gfCNCPoint5[9670] = {X 422.3701, Y 16.1525, Z -7.1667, A 0.000, B 0.000, C 0.000 }
gfCNCPoint5[9671] = {X 421.6779, Y 16.7020, Z -7.1667, A 0.000, B 0.000, C 0.000 }
gfCNCPoint5[9672] = {X 420.8909, Y 17.1044, Z -7.1667, A 0.000, B 0.000, C 0.000 }
gfCNCPoint5[9673] = {X 420.1838, Y 18.0570, Z -7.1667, A 0.000, B 0.000, C 0.000 }
gfCNCPoint5[9674] = {X 419.5438, Y 19.0559, Z -7.1667, A 0.000, B 0.000, C 0.000 }
gfCNCPoint5[9675] = {X 418.0618, Y 21.4548, Z -7.1667, A 0.000, B 0.000, C 0.000 }
gfCNCPoint5[9676] = {X 411.6279, Y 31.7882, Z -7.1667, A 0.000, B 0.000, C 0.000 }
gfCNCPoint5[9677] = {X 411.6285, Y 40.8613, Z -7.1667, A 0.000, B 0.000, C 0.000 }
gfCNCPoint5[9678] = {X 412.2676, Y 41.5581, Z -7.1667, A 0.000, B 0.000, C 0.000 }
gfCNCPoint5[9679] = {X 412.7477, Y 42.3727, Z -7.1667, A 0.000, B 0.000, C 0.000 }
gfCNCPoint5[9680] = {X 413.0478, Y 43.2694, Z -7.1667, A 0.000, B 0.000, C 0.000 }
gfCNCPoint5[9681] = {X 413.1547, Y 44.2088, Z -7.1667, A 0.000, B 0.000, C 0.000 }
gfCNCPoint5[9682] = {X 413.1545, Y 45.0423, Z -7.1667, A 0.000, B 0.000, C 0.000 }
gfCNCPoint5[9683] = {X 413.0719, Y 45.8494, Z -7.1667, A 0.000, B 0.000, C 0.000 }
gfCNCPoint5[9684] = {X 412.8426, Y 46.6276, Z -7.1667, A 0.000, B 0.000, C 0.000 }
gfCNCPoint5[9685] = {X 412.4743, Y 47.3505, Z -7.1667, A 0.000, B 0.000, C 0.000 }
gfCNCPoint5[9686] = {X 411.9795, Y 47.9934, Z -7.1667, A 0.000, B 0.000, C 0.000 }
gfCNCPoint5[9687] = {X 412.3313, Y 48.3200, Z -7.1667, A 0.000, B 0.000, C 0.000 }
gfCNCPoint5[9688] = {X 419.4886, Y 48.3200, Z -7.1667, A 0.000, B 0.000, C 0.000 }
gfCNCPoint5[9689] = {X 420.8006, Y 48.4093, Z -7.1667, A 0.000, B 0.000, C 0.000 }
gfCNCPoint5[9690] = {X 422.0883, Y 48.6756, Z -7.1667, A 0.000, B 0.000, C 0.000 }
gfCNCPoint5[9691] = {X 423.3281, Y 49.1140, Z -7.1667, A 0.000, B 0.000, C 0.000 }
gfCNCPoint5[9692] = {X 424.4970, Y 49.7164, Z -7.1667, A 0.000, B 0.000, C 0.000 }
gfCNCPoint5[9693] = {X 425.4625, Y 50.3832, Z -7.1667, A 0.000, B 0.000, C 0.000 }
gfCNCPoint5[9694] = {X 426.3402, Y 51.1620, Z -7.1667, A 0.000, B 0.000, C 0.000 }
gfCNCPoint5[9695] = {X 427.1172, Y 52.0412, Z -7.1667, A 0.000, B 0.000, C 0.000 }
gfCNCPoint5[9696] = {X 427.7821, Y 53.0080, Z -7.1667, A 0.000, B 0.000, C 0.000 }
gfCNCPoint5[9697] = {X 428.1265, Y 53.6309, Z -7.1667, A 0.000, B 0.000, C 0.000 }
gfCNCPoint5[9698] = {X 428.4242, Y 54.2773, Z -7.1667, A 0.000, B 0.000, C 0.000 }
gfCNCPoint5[9699] = {X 431.5822, Y 55.5078, Z -7.1667, A 0.000, B 0.000, C 0.000 }
gfCNCPoint5[9700] = {X 439.8795, Y 58.7999, Z -7.1667, A 0.000, B 0.000, C 0.000 }
gfCNCPoint5[9701] = {X 441.6498, Y 54.3383, Z -7.1667, A 0.000, B 0.000, C 0.000 }
gfCNCPoint5[9702] = {X 444.2225, Y 55.3591, Z -7.1667, A 0.000, B 0.000, C 0.000 }
gfCNCPoint5[9703] = {X 444.5427, Y 54.0013, Z -7.1667, A 0.000, B 0.000, C 0.000 }
gfCNCPoint5[9704] = {X 444.9921, Y 52.6806, Z -7.1667, A 0.000, B 0.000, C 0.000 }
gfCNCPoint5[9705] = {X 443.9527, Y 53.3760, Z -7.1667, A 0.000, B 0.000, C 0.000 }
gfCNCPoint5[9706] = {X 442.8324, Y 53.9317, Z -7.1667, A 0.000, B 0.000, C 0.000 }
gfCNCPoint5[9707] = {X 441.6498, Y 54.3383, Z -7.1667, A 0.000, B 0.000, C 0.000 }
gfCNCPoint5[9708] = {X 440.7647, Y 56.5691, Z -7.1667, A 0.000, B 0.000, C 0.000 }
gfCNCPoint5[9709] = {X 446.3797, Y 58.7970, Z -7.1667, A 0.000, B 0.000, C 0.000 }
gfCNCPoint5[9710] = {X 446.3796, Y 58.0000, Z -7.1667, A 0.000, B 0.000, C 0.000 }
gfCNCPoint5[9711] = {X 446.4304, Y 56.8937, Z -7.1667, A 0.000, B 0.000, C 0.000 }
gfCNCPoint5[9712] = {X 446.5822, Y 55.7968, Z -7.1667, A 0.000, B 0.000, C 0.000 }
gfCNCPoint5[9713] = {X 446.8494, Y 54.6640, Z -7.1667, A 0.000, B 0.000, C 0.000 }
gfCNCPoint5[9714] = {X 447.2243, Y 53.5622, Z -7.1667, A 0.000, B 0.000, C 0.000 }
gfCNCPoint5[9715] = {X 447.8767, Y 52.1752, Z -7.1667, A 0.000, B 0.000, C 0.000 }
gfCNCPoint5[9716] = {X 448.6995, Y 50.8820, Z -7.1667, A 0.000, B 0.000, C 0.000 }
gfCNCPoint5[9717] = {X 447.8224, Y 50.1272, Z -7.1667, A 0.000, B 0.000, C 0.000 }
gfCNCPoint5[9718] = {X 447.0760, Y 49.2431, Z -7.1667, A 0.000, B 0.000, C 0.000 }
gfCNCPoint5[9719] = {X 446.4792, Y 48.2518, Z -7.1667, A 0.000, B 0.000, C 0.000 }
gfCNCPoint5[9720] = {X 446.0469, Y 47.1785, Z -7.1667, A 0.000, B 0.000, C 0.000 }
gfCNCPoint5[9721] = {X 445.6333, Y 48.2126, Z -7.1667, A 0.000, B 0.000, C 0.000 }
gfCNCPoint5[9722] = {X 445.0668, Y 49.1715, Z -7.1667, A 0.000, B 0.000, C 0.000 }
gfCNCPoint5[9723] = {X 444.3606, Y 50.0328, Z -7.1667, A 0.000, B 0.000, C 0.000 }
gfCNCPoint5[9724] = {X 443.5314, Y 50.7763, Z -7.1667, A 0.000, B 0.000, C 0.000 }
gfCNCPoint5[9725] = {X 442.7497, Y 51.2993, Z -7.1667, A 0.000, B 0.000, C 0.000 }
gfCNCPoint5[9726] = {X 441.9071, Y 51.7172, Z -7.1667, A 0.000, B 0.000, C 0.000 }
gfCNCPoint5[9727] = {X 441.0177, Y 52.0230, Z -7.1667, A 0.000, B 0.000, C 0.000 }
gfCNCPoint5[9728] = {X 440.0677, Y 52.2155, Z -7.1667, A 0.000, B 0.000, C 0.000 }
gfCNCPoint5[9729] = {X 439.1005, Y 52.2800, Z -7.1667, A 0.000, B 0.000, C 0.000 }
gfCNCPoint5[9730] = {X 432.5144, Y 52.2800, Z -7.1667, A 0.000, B 0.000, C 0.000 }
gfCNCPoint5[9731] = {X 431.6034, Y 52.2228, Z -7.1667, A 0.000, B 0.000, C 0.000 }
gfCNCPoint5[9732] = {X 430.7066, Y 52.0520, Z -7.1667, A 0.000, B 0.000, C 0.000 }
gfCNCPoint5[9733] = {X 429.8384, Y 51.7703, Z -7.1667, A 0.000, B 0.000, C 0.000 }
gfCNCPoint5[9734] = {X 430.0166, Y 52.0766, Z -7.1667, A 0.000, B 0.000, C 0.000 }
gfCNCPoint5[9735] = {X 430.1859, Y 52.3880, Z -7.1667, A 0.000, B 0.000, C 0.000 }
gfCNCPoint5[9736] = {X 432.4639, Y 53.2756, Z -7.1667, A 0.000, B 0.000, C 0.000 }
gfCNCPoint5[9737] = {X 440.7647, Y 56.5691, Z -7.1667, A 0.000, B 0.000, C 0.000 }
gfCNCPoint5[9738] = {X 439.8795, Y 58.7999, Z -7.1667, A 0.000, B 0.000, C 0.000 }
gfCNCPoint5[9739] = {X 449.5091, Y 62.6207, Z -7.1667, A 0.000, B 0.000, C 0.000 }
gfCNCPoint5[9740] = {X 449.1112, Y 61.4460, Z -7.1667, A 0.000, B 0.000, C 0.000 }
gfCNCPoint5[9741] = {X 448.8668, Y 60.2301, Z -7.1667, A 0.000, B 0.000, C 0.000 }
gfCNCPoint5[9742] = {X 448.7798, Y 58.9930, Z -7.1667, A 0.000, B 0.000, C 0.000 }
gfCNCPoint5[9743] = {X 448.7796, Y 58.0000, Z -7.1667, A 0.000, B 0.000, C 0.000 }
gfCNCPoint5[9744] = {X 448.8564, Y 56.7833, Z -7.1667, A 0.000, B 0.000, C 0.000 }
gfCNCPoint5[9745] = {X 449.0855, Y 55.5859, Z -7.1667, A 0.000, B 0.000, C 0.000 }
gfCNCPoint5[9746] = {X 449.4632, Y 54.4268, Z -7.1667, A 0.000, B 0.000, C 0.000 }
gfCNCPoint5[9747] = {X 449.9837, Y 53.3244, Z -7.1667, A 0.000, B 0.000, C 0.000 }
gfCNCPoint5[9748] = {X 450.6386, Y 52.2961, Z -7.1667, A 0.000, B 0.000, C 0.000 }
gfCNCPoint5[9749] = {X 451.3887, Y 51.3890, Z -7.1667, A 0.000, B 0.000, C 0.000 }
gfCNCPoint5[9750] = {X 452.2434, Y 50.5796, Z -7.1667, A 0.000, B 0.000, C 0.000 }
gfCNCPoint5[9751] = {X 453.1901, Y 49.8800, Z -7.1667, A 0.000, B 0.000, C 0.000 }
gfCNCPoint5[9752] = {X 452.3731, Y 49.8442, Z -7.1667, A 0.000, B 0.000, C 0.000 }
gfCNCPoint5[9753] = {X 451.5735, Y 49.6724, Z -7.1667, A 0.000, B 0.000, C 0.000 }
gfCNCPoint5[9754] = {X 450.8138, Y 49.3696, Z -7.1667, A 0.000, B 0.000, C 0.000 }
gfCNCPoint5[9755] = {X 450.1154, Y 48.9441, Z -7.1667, A 0.000, B 0.000, C 0.000 }
gfCNCPoint5[9756] = {X 449.3503, Y 48.2496, Z -7.1667, A 0.000, B 0.000, C 0.000 }
gfCNCPoint5[9757] = {X 448.7486, Y 47.4095, Z -7.1667, A 0.000, B 0.000, C 0.000 }
gfCNCPoint5[9758] = {X 448.3373, Y 46.4616, Z -7.1667, A 0.000, B 0.000, C 0.000 }
gfCNCPoint5[9759] = {X 448.1732, Y 45.7588, Z -7.1667, A 0.000, B 0.000, C 0.000 }
gfCNCPoint5[9760] = {X 448.1146, Y 45.0395, Z -7.1667, A 0.000, B 0.000, C 0.000 }
gfCNCPoint5[9761] = {X 448.1149, Y 44.1417, Z -7.1667, A 0.000, B 0.000, C 0.000 }
gfCNCPoint5[9762] = {X 448.2252, Y 43.1751, Z -7.1667, A 0.000, B 0.000, C 0.000 }
gfCNCPoint5[9763] = {X 448.5250, Y 42.2497, Z -7.1667, A 0.000, B 0.000, C 0.000 }
gfCNCPoint5[9764] = {X 449.0024, Y 41.4021, Z -7.1667, A 0.000, B 0.000, C 0.000 }
gfCNCPoint5[9765] = {X 449.6384, Y 40.6660, Z -7.1667, A 0.000, B 0.000, C 0.000 }
gfCNCPoint5[9766] = {X 449.6384, Y 35.0338, Z -7.1667, A 0.000, B 0.000, C 0.000 }
gfCNCPoint5[9767] = {X 447.8174, Y 35.0338, Z -7.1667, A 0.000, B 0.000, C 0.000 }
gfCNCPoint5[9768] = {X 443.7931, Y 42.8695, Z -7.1667, A 0.000, B 0.000, C 0.000 }
gfCNCPoint5[9769] = {X 443.9303, Y 43.5111, Z -7.1667, A 0.000, B 0.000, C 0.000 }
gfCNCPoint5[9770] = {X 443.9803, Y 44.1653, Z -7.1667, A 0.000, B 0.000, C 0.000 }
gfCNCPoint5[9771] = {X 443.9805, Y 45.0000, Z -7.1667, A 0.000, B 0.000, C 0.000 }
gfCNCPoint5[9772] = {X 443.9242, Y 45.7387, Z -7.1667, A 0.000, B 0.000, C 0.000 }
gfCNCPoint5[9773] = {X 443.7568, Y 46.4603, Z -7.1667, A 0.000, B 0.000, C 0.000 }
gfCNCPoint5[9774] = {X 443.3474, Y 47.4038, Z -7.1667, A 0.000, B 0.000, C 0.000 }
gfCNCPoint5[9775] = {X 442.7493, Y 48.2405, Z -7.1667, A 0.000, B 0.000, C 0.000 }
gfCNCPoint5[9776] = {X 441.9891, Y 48.9332, Z -7.1667, A 0.000, B 0.000, C 0.000 }
gfCNCPoint5[9777] = {X 441.1006, Y 49.4513, Z -7.1667, A 0.000, B 0.000, C 0.000 }
gfCNCPoint5[9778] = {X 440.1232, Y 49.7716, Z -7.1667, A 0.000, B 0.000, C 0.000 }
gfCNCPoint5[9779] = {X 439.1005, Y 49.8800, Z -7.1667, A 0.000, B 0.000, C 0.000 }
gfCNCPoint5[9780] = {X 432.5144, Y 49.8800, Z -7.1667, A 0.000, B 0.000, C 0.000 }
gfCNCPoint5[9781] = {X 431.6014, Y 49.7938, Z -7.1667, A 0.000, B 0.000, C 0.000 }
gfCNCPoint5[9782] = {X 430.7206, Y 49.5383, Z -7.1667, A 0.000, B 0.000, C 0.000 }
gfCNCPoint5[9783] = {X 429.8343, Y 49.0782, Z -7.1667, A 0.000, B 0.000, C 0.000 }
gfCNCPoint5[9784] = {X 429.0603, Y 48.4473, Z -7.1667, A 0.000, B 0.000, C 0.000 }
gfCNCPoint5[9785] = {X 428.4309, Y 47.6720, Z -7.1667, A 0.000, B 0.000, C 0.000 }
gfCNCPoint5[9786] = {X 427.9725, Y 46.7848, Z -7.1667, A 0.000, B 0.000, C 0.000 }
gfCNCPoint5[9787] = {X 427.7197, Y 45.9083, Z -7.1667, A 0.000, B 0.000, C 0.000 }
gfCNCPoint5[9788] = {X 427.6344, Y 45.0000, Z -7.1667, A 0.000, B 0.000, C 0.000 }
gfCNCPoint5[9789] = {X 427.6344, Y 44.2089, Z -7.1667, A 0.000, B 0.000, C 0.000 }
gfCNCPoint5[9790] = {X 427.7263, Y 43.2661, Z -7.1667, A 0.000, B 0.000, C 0.000 }
gfCNCPoint5[9791] = {X 427.9987, Y 42.3588, Z -7.1667, A 0.000, B 0.000, C 0.000 }
gfCNCPoint5[9792] = {X 428.4412, Y 41.5212, Z -7.1667, A 0.000, B 0.000, C 0.000 }
gfCNCPoint5[9793] = {X 429.0371, Y 40.7849, Z -7.1667, A 0.000, B 0.000, C 0.000 }
gfCNCPoint5[9794] = {X 429.7641, Y 40.1776, Z -7.1667, A 0.000, B 0.000, C 0.000 }
gfCNCPoint5[9795] = {X 430.5947, Y 39.7222, Z -7.1667, A 0.000, B 0.000, C 0.000 }
gfCNCPoint5[9796] = {X 434.2527, Y 32.5621, Z -7.1667, A 0.000, B 0.000, C 0.000 }
gfCNCPoint5[9797] = {X 432.9253, Y 31.5659, Z -7.1667, A 0.000, B 0.000, C 0.000 }
gfCNCPoint5[9798] = {X 431.7497, Y 30.3944, Z -7.1667, A 0.000, B 0.000, C 0.000 }
gfCNCPoint5[9799] = {X 430.7488, Y 29.0705, Z -7.1667, A 0.000, B 0.000, C 0.000 }
gfCNCPoint5[9800] = {X 429.9422, Y 27.6200, Z -7.1667, A 0.000, B 0.000, C 0.000 }
gfCNCPoint5[9801] = {X 429.3457, Y 26.0712, Z -7.1667, A 0.000, B 0.000, C 0.000 }
gfCNCPoint5[9802] = {X 428.8989, Y 24.1613, Z -7.1667, A 0.000, B 0.000, C 0.000 }
gfCNCPoint5[9803] = {X 428.6737, Y 22.2128, Z -7.1667, A 0.000, B 0.000, C 0.000 }
gfCNCPoint5[9804] = {X 428.6731, Y 20.2514, Z -7.1667, A 0.000, B 0.000, C 0.000 }
gfCNCPoint5[9805] = {X 428.8972, Y 18.3027, Z -7.1667, A 0.000, B 0.000, C 0.000 }
gfCNCPoint5[9806] = {X 429.3429, Y 16.3926, Z -7.1667, A 0.000, B 0.000, C 0.000 }
gfCNCPoint5[9807] = {X 429.8636, Y 14.9601, Z -7.1667, A 0.000, B 0.000, C 0.000 }
gfCNCPoint5[9808] = {X 430.5563, Y 13.6023, Z -7.1667, A 0.000, B 0.000, C 0.000 }
gfCNCPoint5[9809] = {X 431.4105, Y 12.3399, Z -7.1667, A 0.000, B 0.000, C 0.000 }
gfCNCPoint5[9810] = {X 432.4132, Y 11.1919, Z -7.1667, A 0.000, B 0.000, C 0.000 }
gfCNCPoint5[9811] = {X 433.5448, Y 10.1793, Z -7.1667, A 0.000, B 0.000, C 0.000 }
gfCNCPoint5[9812] = {X 434.7918, Y 9.3127, Z -7.1667, A 0.000, B 0.000, C 0.000 }
gfCNCPoint5[9813] = {X 436.1354, Y 8.6052, Z -7.1667, A 0.000, B 0.000, C 0.000 }
gfCNCPoint5[9814] = {X 437.5555, Y 8.0674, Z -7.1667, A 0.000, B 0.000, C 0.000 }
gfCNCPoint5[9815] = {X 439.0308, Y 7.7073, Z -7.1667, A 0.000, B 0.000, C 0.000 }
gfCNCPoint5[9816] = {X 441.1775, Y 7.4101, Z -7.1667, A 0.000, B 0.000, C 0.000 }
gfCNCPoint5[9817] = {X 443.3425, Y 7.3136, Z -7.1667, A 0.000, B 0.000, C 0.000 }
gfCNCPoint5[9818] = {X 459.4469, Y 7.3096, Z -7.1667, A 0.000, B 0.000, C 0.000 }
gfCNCPoint5[9819] = {X 460.4098, Y 7.4057, Z -7.1667, A 0.000, B 0.000, C 0.000 }
gfCNCPoint5[9820] = {X 461.3347, Y 7.6903, Z -7.1667, A 0.000, B 0.000, C 0.000 }
gfCNCPoint5[9821] = {X 462.1851, Y 8.1521, Z -7.1667, A 0.000, B 0.000, C 0.000 }
gfCNCPoint5[9822] = {X 462.9274, Y 8.7728, Z -7.1667, A 0.000, B 0.000, C 0.000 }
gfCNCPoint5[9823] = {X 463.5324, Y 9.5281, Z -7.1667, A 0.000, B 0.000, C 0.000 }
gfCNCPoint5[9824] = {X 463.9761, Y 10.3881, Z -7.1667, A 0.000, B 0.000, C 0.000 }
gfCNCPoint5[9825] = {X 464.2317, Y 11.2682, Z -7.1667, A 0.000, B 0.000, C 0.000 }
gfCNCPoint5[9826] = {X 464.3179, Y 12.1806, Z -7.1667, A 0.000, B 0.000, C 0.000 }
gfCNCPoint5[9827] = {X 464.3179, Y 12.9780, Z -7.1667, A 0.000, B 0.000, C 0.000 }
gfCNCPoint5[9828] = {X 464.2174, Y 13.9633, Z -7.1667, A 0.000, B 0.000, C 0.000 }
gfCNCPoint5[9829] = {X 463.9200, Y 14.9081, Z -7.1667, A 0.000, B 0.000, C 0.000 }
gfCNCPoint5[9830] = {X 463.4380, Y 15.7733, Z -7.1667, A 0.000, B 0.000, C 0.000 }
gfCNCPoint5[9831] = {X 462.7912, Y 16.5234, Z -7.1667, A 0.000, B 0.000, C 0.000 }
gfCNCPoint5[9832] = {X 462.7910, Y 16.7696, Z -7.1667, A 0.000, B 0.000, C 0.000 }
gfCNCPoint5[9833] = {X 462.7919, Y 40.6641, Z -7.1667, A 0.000, B 0.000, C 0.000 }
gfCNCPoint5[9834] = {X 463.4324, Y 41.4055, Z -7.1667, A 0.000, B 0.000, C 0.000 }
gfCNCPoint5[9835] = {X 463.9119, Y 42.2600, Z -7.1667, A 0.000, B 0.000, C 0.000 }
gfCNCPoint5[9836] = {X 464.2110, Y 43.1930, Z -7.1667, A 0.000, B 0.000, C 0.000 }
gfCNCPoint5[9837] = {X 464.3178, Y 44.1670, Z -7.1667, A 0.000, B 0.000, C 0.000 }
gfCNCPoint5[9838] = {X 464.3179, Y 45.0000, Z -7.1667, A 0.000, B 0.000, C 0.000 }
gfCNCPoint5[9839] = {X 464.3082, Y 45.3090, Z -7.1667, A 0.000, B 0.000, C 0.000 }
gfCNCPoint5[9840] = {X 464.2788, Y 45.6167, Z -7.1667, A 0.000, B 0.000, C 0.000 }
gfCNCPoint5[9841] = {X 464.0485, Y 46.5992, Z -7.1667, A 0.000, B 0.000, C 0.000 }
gfCNCPoint5[9842] = {X 463.6209, Y 47.5134, Z -7.1667, A 0.000, B 0.000, C 0.000 }
gfCNCPoint5[9843] = {X 463.0145, Y 48.3200, Z -7.1667, A 0.000, B 0.000, C 0.000 }
gfCNCPoint5[9844] = {X 462.6627, Y 47.9934, Z -7.1667, A 0.000, B 0.000, C 0.000 }
gfCNCPoint5[9845] = {X 461.9835, Y 48.5889, Z -7.1667, A 0.000, B 0.000, C 0.000 }
gfCNCPoint5[9846] = {X 461.1970, Y 49.0331, Z -7.1667, A 0.000, B 0.000, C 0.000 }
gfCNCPoint5[9847] = {X 460.3364, Y 49.3073, Z -7.1667, A 0.000, B 0.000, C 0.000 }
gfCNCPoint5[9848] = {X 459.4379, Y 49.4000, Z -7.1667, A 0.000, B 0.000, C 0.000 }
gfCNCPoint5[9849] = {X 452.9945, Y 49.4000, Z -7.1667, A 0.000, B 0.000, C 0.000 }
gfCNCPoint5[9850] = {X 452.0154, Y 49.2897, Z -7.1667, A 0.000, B 0.000, C 0.000 }
gfCNCPoint5[9851] = {X 451.0854, Y 48.9643, Z -7.1667, A 0.000, B 0.000, C 0.000 }
gfCNCPoint5[9852] = {X 450.2511, Y 48.4400, Z -7.1667, A 0.000, B 0.000, C 0.000 }
gfCNCPoint5[9853] = {X 449.5544, Y 47.7433, Z -7.1667, A 0.000, B 0.000, C 0.000 }
gfCNCPoint5[9854] = {X 449.0302, Y 46.9091, Z -7.1667, A 0.000, B 0.000, C 0.000 }
gfCNCPoint5[9855] = {X 448.7048, Y 45.9791, Z -7.1667, A 0.000, B 0.000, C 0.000 }
gfCNCPoint5[9856] = {X 448.5945, Y 45.0000, Z -7.1667, A 0.000, B 0.000, C 0.000 }
gfCNCPoint5[9857] = {X 448.5949, Y 44.1483, Z -7.1667, A 0.000, B 0.000, C 0.000 }
gfCNCPoint5[9858] = {X 448.7053, Y 43.2275, Z -7.1667, A 0.000, B 0.000, C 0.000 }
gfCNCPoint5[9859] = {X 449.0063, Y 42.3503, Z -7.1667, A 0.000, B 0.000, C 0.000 }
gfCNCPoint5[9860] = {X 449.4844, Y 41.5556, Z -7.1667, A 0.000, B 0.000, C 0.000 }
gfCNCPoint5[9861] = {X 450.1184, Y 40.8789, Z -7.1667, A 0.000, B 0.000, C 0.000 }
gfCNCPoint5[9862] = {X 450.1184, Y 34.5538, Z -7.1667, A 0.000, B 0.000, C 0.000 }
gfCNCPoint5[9863] = {X 447.5243, Y 34.5538, Z -7.1667, A 0.000, B 0.000, C 0.000 }
gfCNCPoint5[9864] = {X 443.2769, Y 42.8240, Z -7.1667, A 0.000, B 0.000, C 0.000 }
gfCNCPoint5[9865] = {X 443.4442, Y 43.5075, Z -7.1667, A 0.000, B 0.000, C 0.000 }
gfCNCPoint5[9866] = {X 443.5005, Y 44.2089, Z -7.1667, A 0.000, B 0.000, C 0.000 }
gfCNCPoint5[9867] = {X 443.5005, Y 45.0000, Z -7.1667, A 0.000, B 0.000, C 0.000 }
gfCNCPoint5[9868] = {X 443.3902, Y 45.9791, Z -7.1667, A 0.000, B 0.000, C 0.000 }
gfCNCPoint5[9869] = {X 443.0647, Y 46.9091, Z -7.1667, A 0.000, B 0.000, C 0.000 }
gfCNCPoint5[9870] = {X 442.5405, Y 47.7434, Z -7.1667, A 0.000, B 0.000, C 0.000 }
gfCNCPoint5[9871] = {X 441.8438, Y 48.4401, Z -7.1667, A 0.000, B 0.000, C 0.000 }
gfCNCPoint5[9872] = {X 441.0096, Y 48.9643, Z -7.1667, A 0.000, B 0.000, C 0.000 }
gfCNCPoint5[9873] = {X 440.0796, Y 49.2897, Z -7.1667, A 0.000, B 0.000, C 0.000 }
gfCNCPoint5[9874] = {X 439.1005, Y 49.4000, Z -7.1667, A 0.000, B 0.000, C 0.000 }
gfCNCPoint5[9875] = {X 432.5144, Y 49.4000, Z -7.1667, A 0.000, B 0.000, C 0.000 }
gfCNCPoint5[9876] = {X 431.5353, Y 49.2897, Z -7.1667, A 0.000, B 0.000, C 0.000 }
gfCNCPoint5[9877] = {X 430.6053, Y 48.9643, Z -7.1667, A 0.000, B 0.000, C 0.000 }
gfCNCPoint5[9878] = {X 429.7711, Y 48.4401, Z -7.1667, A 0.000, B 0.000, C 0.000 }
gfCNCPoint5[9879] = {X 429.0743, Y 47.7434, Z -7.1667, A 0.000, B 0.000, C 0.000 }
gfCNCPoint5[9880] = {X 428.5501, Y 46.9091, Z -7.1667, A 0.000, B 0.000, C 0.000 }
gfCNCPoint5[9881] = {X 428.2247, Y 45.9791, Z -7.1667, A 0.000, B 0.000, C 0.000 }
gfCNCPoint5[9882] = {X 428.1144, Y 45.0000, Z -7.1667, A 0.000, B 0.000, C 0.000 }
gfCNCPoint5[9883] = {X 428.1148, Y 44.1483, Z -7.1667, A 0.000, B 0.000, C 0.000 }
gfCNCPoint5[9884] = {X 428.2132, Y 43.2816, Z -7.1667, A 0.000, B 0.000, C 0.000 }
gfCNCPoint5[9885] = {X 428.4806, Y 42.4514, Z -7.1667, A 0.000, B 0.000, C 0.000 }
gfCNCPoint5[9886] = {X 428.9065, Y 41.6903, Z -7.1667, A 0.000, B 0.000, C 0.000 }
gfCNCPoint5[9887] = {X 429.4741, Y 41.0281, Z -7.1667, A 0.000, B 0.000, C 0.000 }
gfCNCPoint5[9888] = {X 430.1613, Y 40.4909, Z -7.1667, A 0.000, B 0.000, C 0.000 }
gfCNCPoint5[9889] = {X 430.9408, Y 40.0998, Z -7.1667, A 0.000, B 0.000, C 0.000 }
gfCNCPoint5[9890] = {X 434.8812, Y 32.3870, Z -7.1667, A 0.000, B 0.000, C 0.000 }
gfCNCPoint5[9891] = {X 433.7234, Y 31.5994, Z -7.1667, A 0.000, B 0.000, C 0.000 }
gfCNCPoint5[9892] = {X 432.6710, Y 30.6758, Z -7.1667, A 0.000, B 0.000, C 0.000 }
gfCNCPoint5[9893] = {X 431.7398, Y 29.6301, Z -7.1667, A 0.000, B 0.000, C 0.000 }
gfCNCPoint5[9894] = {X 430.9438, Y 28.4781, Z -7.1667, A 0.000, B 0.000, C 0.000 }
gfCNCPoint5[9895] = {X 430.2950, Y 27.2372, Z -7.1667, A 0.000, B 0.000, C 0.000 }
gfCNCPoint5[9896] = {X 429.8033, Y 25.9262, Z -7.1667, A 0.000, B 0.000, C 0.000 }
gfCNCPoint5[9897] = {X 429.3704, Y 24.0715, Z -7.1667, A 0.000, B 0.000, C 0.000 }
gfCNCPoint5[9898] = {X 429.1525, Y 22.1795, Z -7.1667, A 0.000, B 0.000, C 0.000 }
gfCNCPoint5[9899] = {X 429.1525, Y 20.2750, Z -7.1667, A 0.000, B 0.000, C 0.000 }
gfCNCPoint5[9900] = {X 429.3704, Y 18.3830, Z -7.1667, A 0.000, B 0.000, C 0.000 }
gfCNCPoint5[9901] = {X 429.8033, Y 16.5283, Z -7.1667, A 0.000, B 0.000, C 0.000 }
gfCNCPoint5[9902] = {X 430.3769, Y 14.9868, Z -7.1667, A 0.000, B 0.000, C 0.000 }
gfCNCPoint5[9903] = {X 431.1574, Y 13.5390, Z -7.1667, A 0.000, B 0.000, C 0.000 }
gfCNCPoint5[9904] = {X 432.1300, Y 12.2125, Z -7.1667, A 0.000, B 0.000, C 0.000 }
gfCNCPoint5[9905] = {X 433.2760, Y 11.0327, Z -7.1667, A 0.000, B 0.000, C 0.000 }
gfCNCPoint5[9906] = {X 434.5736, Y 10.0220, Z -7.1667, A 0.000, B 0.000, C 0.000 }
gfCNCPoint5[9907] = {X 435.9982, Y 9.1998, Z -7.1667, A 0.000, B 0.000, C 0.000 }
gfCNCPoint5[9908] = {X 437.5224, Y 8.5817, Z -7.1667, A 0.000, B 0.000, C 0.000 }
gfCNCPoint5[9909] = {X 439.1172, Y 8.1795, Z -7.1667, A 0.000, B 0.000, C 0.000 }
gfCNCPoint5[9910] = {X 441.2213, Y 7.8881, Z -7.1667, A 0.000, B 0.000, C 0.000 }
gfCNCPoint5[9911] = {X 443.3434, Y 7.7936, Z -7.1667, A 0.000, B 0.000, C 0.000 }
gfCNCPoint5[9912] = {X 444.0367, Y 7.7896, Z -7.1667, A 0.000, B 0.000, C 0.000 }
gfCNCPoint5[9913] = {X 459.4469, Y 7.7896, Z -7.1667, A 0.000, B 0.000, C 0.000 }
gfCNCPoint5[9914] = {X 460.4240, Y 7.8997, Z -7.1667, A 0.000, B 0.000, C 0.000 }
gfCNCPoint5[9915] = {X 461.3521, Y 8.2244, Z -7.1667, A 0.000, B 0.000, C 0.000 }
gfCNCPoint5[9916] = {X 462.1847, Y 8.7476, Z -7.1667, A 0.000, B 0.000, C 0.000 }
gfCNCPoint5[9917] = {X 462.8799, Y 9.4429, Z -7.1667, A 0.000, B 0.000, C 0.000 }
gfCNCPoint5[9918] = {X 463.4031, Y 10.2754, Z -7.1667, A 0.000, B 0.000, C 0.000 }
gfCNCPoint5[9919] = {X 463.7278, Y 11.2035, Z -7.1667, A 0.000, B 0.000, C 0.000 }
gfCNCPoint5[9920] = {X 463.8379, Y 12.1806, Z -7.1667, A 0.000, B 0.000, C 0.000 }
gfCNCPoint5[9921] = {X 463.8377, Y 13.0201, Z -7.1667, A 0.000, B 0.000, C 0.000 }
gfCNCPoint5[9922] = {X 463.7300, Y 13.9467, Z -7.1667, A 0.000, B 0.000, C 0.000 }
gfCNCPoint5[9923] = {X 463.4293, Y 14.8297, Z -7.1667, A 0.000, B 0.000, C 0.000 }
gfCNCPoint5[9924] = {X 462.9493, Y 15.6295, Z -7.1667, A 0.000, B 0.000, C 0.000 }
gfCNCPoint5[9925] = {X 462.3114, Y 16.3102, Z -7.1667, A 0.000, B 0.000, C 0.000 }
gfCNCPoint5[9926] = {X 462.3110, Y 16.7691, Z -7.1667, A 0.000, B 0.000, C 0.000 }
gfCNCPoint5[9927] = {X 462.3119, Y 40.8771, Z -7.1667, A 0.000, B 0.000, C 0.000 }
gfCNCPoint5[9928] = {X 462.9559, Y 41.5661, Z -7.1667, A 0.000, B 0.000, C 0.000 }
gfCNCPoint5[9929] = {X 463.4383, Y 42.3766, Z -7.1667, A 0.000, B 0.000, C 0.000 }
gfCNCPoint5[9930] = {X 463.7369, Y 43.2712, Z -7.1667, A 0.000, B 0.000, C 0.000 }
gfCNCPoint5[9931] = {X 463.8379, Y 44.2088, Z -7.1667, A 0.000, B 0.000, C 0.000 }
gfCNCPoint5[9932] = {X 463.8379, Y 45.0000, Z -7.1667, A 0.000, B 0.000, C 0.000 }
gfCNCPoint5[9933] = {X 463.7612, Y 45.8182, Z -7.1667, A 0.000, B 0.000, C 0.000 }
gfCNCPoint5[9934] = {X 463.5336, Y 46.6079, Z -7.1667, A 0.000, B 0.000, C 0.000 }
gfCNCPoint5[9935] = {X 463.1632, Y 47.3415, Z -7.1667, A 0.000, B 0.000, C 0.000 }
gfCNCPoint5[9936] = {X 462.6627, Y 47.9934, Z -7.1667, A 0.000, B 0.000, C 0.000 }
gfCNCPoint5[9937] = {X 463.0145, Y 48.3200, Z -7.1667, A 0.000, B 0.000, C 0.000 }
gfCNCPoint5[9938] = {X 472.1884, Y 48.3200, Z -7.1667, A 0.000, B 0.000, C 0.000 }
gfCNCPoint5[9939] = {X 471.5820, Y 47.5134, Z -7.1667, A 0.000, B 0.000, C 0.000 }
gfCNCPoint5[9940] = {X 471.1544, Y 46.5992, Z -7.1667, A 0.000, B 0.000, C 0.000 }
gfCNCPoint5[9941] = {X 470.9241, Y 45.6167, Z -7.1667, A 0.000, B 0.000, C 0.000 }
gfCNCPoint5[9942] = {X 470.8947, Y 45.3090, Z -7.1667, A 0.000, B 0.000, C 0.000 }
gfCNCPoint5[9943] = {X 470.8850, Y 45.0000, Z -7.1667, A 0.000, B 0.000, C 0.000 }
gfCNCPoint5[9944] = {X 470.8850, Y 44.2089, Z -7.1667, A 0.000, B 0.000, C 0.000 }
gfCNCPoint5[9945] = {X 470.9769, Y 43.2661, Z -7.1667, A 0.000, B 0.000, C 0.000 }
gfCNCPoint5[9946] = {X 471.2492, Y 42.3588, Z -7.1667, A 0.000, B 0.000, C 0.000 }
gfCNCPoint5[9947] = {X 471.6917, Y 41.5212, Z -7.1667, A 0.000, B 0.000, C 0.000 }
gfCNCPoint5[9948] = {X 472.2877, Y 40.7849, Z -7.1667, A 0.000, B 0.000, C 0.000 }
gfCNCPoint5[9949] = {X 473.0147, Y 40.1776, Z -7.1667, A 0.000, B 0.000, C 0.000 }
gfCNCPoint5[9950] = {X 473.8453, Y 39.7222, Z -7.1667, A 0.000, B 0.000, C 0.000 }
gfCNCPoint5[9951] = {X 477.5001, Y 32.5684, Z -7.1667, A 0.000, B 0.000, C 0.000 }
gfCNCPoint5[9952] = {X 476.2821, Y 31.6589, Z -7.1667, A 0.000, B 0.000, C 0.000 }
gfCNCPoint5[9953] = {X 475.1887, Y 30.6028, Z -7.1667, A 0.000, B 0.000, C 0.000 }
gfCNCPoint5[9954] = {X 474.2374, Y 29.4172, Z -7.1667, A 0.000, B 0.000, C 0.000 }
gfCNCPoint5[9955] = {X 473.4434, Y 28.1209, Z -7.1667, A 0.000, B 0.000, C 0.000 }
gfCNCPoint5[9956] = {X 472.8195, Y 26.7347, Z -7.1667, A 0.000, B 0.000, C 0.000 }
gfCNCPoint5[9957] = {X 472.3757, Y 25.2808, Z -7.1667, A 0.000, B 0.000, C 0.000 }
gfCNCPoint5[9958] = {X 472.0516, Y 23.5416, Z -7.1667, A 0.000, B 0.000, C 0.000 }
gfCNCPoint5[9959] = {X 471.9067, Y 21.7784, Z -7.1667, A 0.000, B 0.000, C 0.000 }
gfCNCPoint5[9960] = {X 471.9426, Y 20.0095, Z -7.1667, A 0.000, B 0.000, C 0.000 }
gfCNCPoint5[9961] = {X 472.1589, Y 18.2536, Z -7.1667, A 0.000, B 0.000, C 0.000 }
gfCNCPoint5[9962] = {X 472.5533, Y 16.5290, Z -7.1667, A 0.000, B 0.000, C 0.000 }
gfCNCPoint5[9963] = {X 473.0721, Y 15.0579, Z -7.1667, A 0.000, B 0.000, C 0.000 }
gfCNCPoint5[9964] = {X 473.7716, Y 13.6637, Z -7.1667, A 0.000, B 0.000, C 0.000 }
gfCNCPoint5[9965] = {X 474.6406, Y 12.3684, Z -7.1667, A 0.000, B 0.000, C 0.000 }
gfCNCPoint5[9966] = {X 475.6655, Y 11.1924, Z -7.1667, A 0.000, B 0.000, C 0.000 }
gfCNCPoint5[9967] = {X 476.7430, Y 10.2232, Z -7.1667, A 0.000, B 0.000, C 0.000 }
gfCNCPoint5[9968] = {X 477.9264, Y 9.3865, Z -7.1667, A 0.000, B 0.000, C 0.000 }
gfCNCPoint5[9969] = {X 479.1993, Y 8.6936, Z -7.1667, A 0.000, B 0.000, C 0.000 }
gfCNCPoint5[9970] = {X 480.5444, Y 8.1540, Z -7.1667, A 0.000, B 0.000, C 0.000 }
gfCNCPoint5[9971] = {X 481.9433, Y 7.7751, Z -7.1667, A 0.000, B 0.000, C 0.000 }
gfCNCPoint5[9972] = {X 484.0946, Y 7.4401, Z -7.1667, A 0.000, B 0.000, C 0.000 }
gfCNCPoint5[9973] = {X 486.2686, Y 7.3218, Z -7.1667, A 0.000, B 0.000, C 0.000 }
gfCNCPoint5[9974] = {X 486.9707, Y 7.3096, Z -7.1667, A 0.000, B 0.000, C 0.000 }
gfCNCPoint5[9975] = {X 502.2122, Y 7.3096, Z -7.1667, A 0.000, B 0.000, C 0.000 }
gfCNCPoint5[9976] = {X 502.7438, Y 7.3137, Z -7.1667, A 0.000, B 0.000, C 0.000 }
gfCNCPoint5[9977] = {X 503.6983, Y 7.4159, Z -7.1667, A 0.000, B 0.000, C 0.000 }
gfCNCPoint5[9978] = {X 504.6140, Y 7.7036, Z -7.1667, A 0.000, B 0.000, C 0.000 }
gfCNCPoint5[9979] = {X 505.4554, Y 8.1656, Z -7.1667, A 0.000, B 0.000, C 0.000 }
gfCNCPoint5[9980] = {X 506.1897, Y 8.7838, Z -7.1667, A 0.000, B 0.000, C 0.000 }
gfCNCPoint5[9981] = {X 506.7882, Y 9.5343, Z -7.1667, A 0.000, B 0.000, C 0.000 }
gfCNCPoint5[9982] = {X 507.2276, Y 10.3876, Z -7.1667, A 0.000, B 0.000, C 0.000 }
gfCNCPoint5[9983] = {X 507.4825, Y 11.2658, Z -7.1667, A 0.000, B 0.000, C 0.000 }
gfCNCPoint5[9984] = {X 507.5685, Y 12.1762, Z -7.1667, A 0.000, B 0.000, C 0.000 }
gfCNCPoint5[9985] = {X 507.5683, Y 13.0237, Z -7.1667, A 0.000, B 0.000, C 0.000 }
gfCNCPoint5[9986] = {X 507.4609, Y 13.9969, Z -7.1667, A 0.000, B 0.000, C 0.000 }
gfCNCPoint5[9987] = {X 507.1615, Y 14.9290, Z -7.1667, A 0.000, B 0.000, C 0.000 }
gfCNCPoint5[9988] = {X 506.6820, Y 15.7827, Z -7.1667, A 0.000, B 0.000, C 0.000 }
gfCNCPoint5[9989] = {X 506.0418, Y 16.5234, Z -7.1667, A 0.000, B 0.000, C 0.000 }
gfCNCPoint5[9990] = {X 506.0420, Y 40.6636, Z -7.1667, A 0.000, B 0.000, C 0.000 }
gfCNCPoint5[9991] = {X 506.6827, Y 41.4050, Z -7.1667, A 0.000, B 0.000, C 0.000 }
gfCNCPoint5[9992] = {X 507.1623, Y 42.2595, Z -7.1667, A 0.000, B 0.000, C 0.000 }
gfCNCPoint5[9993] = {X 507.4615, Y 43.1925, Z -7.1667, A 0.000, B 0.000, C 0.000 }
gfCNCPoint5[9994] = {X 507.5683, Y 44.1665, Z -7.1667, A 0.000, B 0.000, C 0.000 }
gfCNCPoint5[9995] = {X 507.5685, Y 45.0000, Z -7.1667, A 0.000, B 0.000, C 0.000 }
gfCNCPoint5[9996] = {X 507.4747, Y 45.9520, Z -7.1667, A 0.000, B 0.000, C 0.000 }
gfCNCPoint5[9997] = {X 507.1970, Y 46.8675, Z -7.1667, A 0.000, B 0.000, C 0.000 }
gfCNCPoint5[9998] = {X 506.7461, Y 47.7112, Z -7.1667, A 0.000, B 0.000, C 0.000 }
gfCNCPoint5[9999] = {X 506.1392, Y 48.4507, Z -7.1667, A 0.000, B 0.000, C 0.000 }
gfCNCPoint5[10000] = {X 505.3997, Y 49.0576, Z -7.1667, A 0.000, B 0.000, C 0.000 }
gfCNCPoint5[10001] = {X 504.5560, Y 49.5085, Z -7.1667, A 0.000, B 0.000, C 0.000 }
gfCNCPoint5[10002] = {X 503.6405, Y 49.7862, Z -7.1667, A 0.000, B 0.000, C 0.000 }
gfCNCPoint5[10003] = {X 502.6885, Y 49.8800, Z -7.1667, A 0.000, B 0.000, C 0.000 }
gfCNCPoint5[10004] = {X 496.2450, Y 49.8800, Z -7.1667, A 0.000, B 0.000, C 0.000 }
gfCNCPoint5[10005] = {X 495.2220, Y 49.7716, Z -7.1667, A 0.000, B 0.000, C 0.000 }
gfCNCPoint5[10006] = {X 494.2445, Y 49.4511, Z -7.1667, A 0.000, B 0.000, C 0.000 }
gfCNCPoint5[10007] = {X 493.3559, Y 48.9328, Z -7.1667, A 0.000, B 0.000, C 0.000 }
gfCNCPoint5[10008] = {X 492.5956, Y 48.2398, Z -7.1667, A 0.000, B 0.000, C 0.000 }
gfCNCPoint5[10009] = {X 491.9976, Y 47.4028, Z -7.1667, A 0.000, B 0.000, C 0.000 }
gfCNCPoint5[10010] = {X 491.5882, Y 46.4590, Z -7.1667, A 0.000, B 0.000, C 0.000 }
gfCNCPoint5[10011] = {X 491.4241, Y 45.7570, Z -7.1667, A 0.000, B 0.000, C 0.000 }
gfCNCPoint5[10012] = {X 491.3652, Y 45.0385, Z -7.1667, A 0.000, B 0.000, C 0.000 }
gfCNCPoint5[10013] = {X 491.3655, Y 44.1417, Z -7.1667, A 0.000, B 0.000, C 0.000 }
gfCNCPoint5[10014] = {X 491.4758, Y 43.1751, Z -7.1667, A 0.000, B 0.000, C 0.000 }
gfCNCPoint5[10015] = {X 491.7755, Y 42.2497, Z -7.1667, A 0.000, B 0.000, C 0.000 }
gfCNCPoint5[10016] = {X 492.2530, Y 41.4021, Z -7.1667, A 0.000, B 0.000, C 0.000 }
gfCNCPoint5[10017] = {X 492.8890, Y 40.6660, Z -7.1667, A 0.000, B 0.000, C 0.000 }
gfCNCPoint5[10018] = {X 492.8890, Y 35.0338, Z -7.1667, A 0.000, B 0.000, C 0.000 }
gfCNCPoint5[10019] = {X 491.0674, Y 35.0338, Z -7.1667, A 0.000, B 0.000, C 0.000 }
gfCNCPoint5[10020] = {X 487.0436, Y 42.8695, Z -7.1667, A 0.000, B 0.000, C 0.000 }
gfCNCPoint5[10021] = {X 487.1809, Y 43.5109, Z -7.1667, A 0.000, B 0.000, C 0.000 }
gfCNCPoint5[10022] = {X 487.2308, Y 44.1648, Z -7.1667, A 0.000, B 0.000, C 0.000 }
gfCNCPoint5[10023] = {X 487.2310, Y 45.0000, Z -7.1667, A 0.000, B 0.000, C 0.000 }
gfCNCPoint5[10024] = {X 487.1749, Y 45.7380, Z -7.1667, A 0.000, B 0.000, C 0.000 }
gfCNCPoint5[10025] = {X 487.0078, Y 46.4590, Z -7.1667, A 0.000, B 0.000, C 0.000 }
gfCNCPoint5[10026] = {X 486.5939, Y 47.4110, Z -7.1667, A 0.000, B 0.000, C 0.000 }
gfCNCPoint5[10027] = {X 485.9879, Y 48.2538, Z -7.1667, A 0.000, B 0.000, C 0.000 }
gfCNCPoint5[10028] = {X 485.2175, Y 48.9494, Z -7.1667, A 0.000, B 0.000, C 0.000 }
gfCNCPoint5[10029] = {X 484.3173, Y 49.4663, Z -7.1667, A 0.000, B 0.000, C 0.000 }
gfCNCPoint5[10030] = {X 483.3557, Y 49.7755, Z -7.1667, A 0.000, B 0.000, C 0.000 }
gfCNCPoint5[10031] = {X 482.3510, Y 49.8800, Z -7.1667, A 0.000, B 0.000, C 0.000 }
gfCNCPoint5[10032] = {X 480.2695, Y 49.8800, Z -7.1667, A 0.000, B 0.000, C 0.000 }
gfCNCPoint5[10033] = {X 480.2695, Y 49.4000, Z -7.1667, A 0.000, B 0.000, C 0.000 }
gfCNCPoint5[10034] = {X 475.7650, Y 49.4000, Z -7.1667, A 0.000, B 0.000, C 0.000 }
gfCNCPoint5[10035] = {X 474.7859, Y 49.2897, Z -7.1667, A 0.000, B 0.000, C 0.000 }
gfCNCPoint5[10036] = {X 473.8559, Y 48.9643, Z -7.1667, A 0.000, B 0.000, C 0.000 }
gfCNCPoint5[10037] = {X 473.0216, Y 48.4401, Z -7.1667, A 0.000, B 0.000, C 0.000 }
gfCNCPoint5[10038] = {X 472.3249, Y 47.7434, Z -7.1667, A 0.000, B 0.000, C 0.000 }
gfCNCPoint5[10039] = {X 471.8007, Y 46.9091, Z -7.1667, A 0.000, B 0.000, C 0.000 }
gfCNCPoint5[10040] = {X 471.4753, Y 45.9791, Z -7.1667, A 0.000, B 0.000, C 0.000 }
gfCNCPoint5[10041] = {X 471.3650, Y 45.0000, Z -7.1667, A 0.000, B 0.000, C 0.000 }
gfCNCPoint5[10042] = {X 471.3654, Y 44.1483, Z -7.1667, A 0.000, B 0.000, C 0.000 }
gfCNCPoint5[10043] = {X 471.4638, Y 43.2816, Z -7.1667, A 0.000, B 0.000, C 0.000 }
gfCNCPoint5[10044] = {X 471.7311, Y 42.4514, Z -7.1667, A 0.000, B 0.000, C 0.000 }
gfCNCPoint5[10045] = {X 472.1570, Y 41.6903, Z -7.1667, A 0.000, B 0.000, C 0.000 }
gfCNCPoint5[10046] = {X 472.7247, Y 41.0281, Z -7.1667, A 0.000, B 0.000, C 0.000 }
gfCNCPoint5[10047] = {X 473.4118, Y 40.4909, Z -7.1667, A 0.000, B 0.000, C 0.000 }
gfCNCPoint5[10048] = {X 474.1914, Y 40.0998, Z -7.1667, A 0.000, B 0.000, C 0.000 }
gfCNCPoint5[10049] = {X 478.1276, Y 32.3951, Z -7.1667, A 0.000, B 0.000, C 0.000 }
gfCNCPoint5[10050] = {X 476.8701, Y 31.5215, Z -7.1667, A 0.000, B 0.000, C 0.000 }
gfCNCPoint5[10051] = {X 475.7394, Y 30.4891, Z -7.1667, A 0.000, B 0.000, C 0.000 }
gfCNCPoint5[10052] = {X 474.7554, Y 29.3159, Z -7.1667, A 0.000, B 0.000, C 0.000 }
gfCNCPoint5[10053] = {X 473.9355, Y 28.0228, Z -7.1667, A 0.000, B 0.000, C 0.000 }
gfCNCPoint5[10054] = {X 473.2941, Y 26.6325, Z -7.1667, A 0.000, B 0.000, C 0.000 }
gfCNCPoint5[10055] = {X 472.8426, Y 25.1694, Z -7.1667, A 0.000, B 0.000, C 0.000 }
gfCNCPoint5[10056] = {X 472.5274, Y 23.4783, Z -7.1667, A 0.000, B 0.000, C 0.000 }
gfCNCPoint5[10057] = {X 472.3865, Y 21.7639, Z -7.1667, A 0.000, B 0.000, C 0.000 }
gfCNCPoint5[10058] = {X 472.4214, Y 20.0440, Z -7.1667, A 0.000, B 0.000, C 0.000 }
gfCNCPoint5[10059] = {X 472.6317, Y 18.3367, Z -7.1667, A 0.000, B 0.000, C 0.000 }
gfCNCPoint5[10060] = {X 473.0152, Y 16.6597, Z -7.1667, A 0.000, B 0.000, C 0.000 }
gfCNCPoint5[10061] = {X 473.5618, Y 15.1345, Z -7.1667, A 0.000, B 0.000, C 0.000 }
gfCNCPoint5[10062] = {X 474.3104, Y 13.6975, Z -7.1667, A 0.000, B 0.000, C 0.000 }
gfCNCPoint5[10063] = {X 475.2470, Y 12.3754, Z -7.1667, A 0.000, B 0.000, C 0.000 }
gfCNCPoint5[10064] = {X 476.3543, Y 11.1925, Z -7.1667, A 0.000, B 0.000, C 0.000 }
gfCNCPoint5[10065] = {X 477.6118, Y 10.1708, Z -7.1667, A 0.000, B 0.000, C 0.000 }
gfCNCPoint5[10066] = {X 478.9963, Y 9.3292, Z -7.1667, A 0.000, B 0.000, C 0.000 }
gfCNCPoint5[10067] = {X 480.4823, Y 8.6832, Z -7.1667, A 0.000, B 0.000, C 0.000 }
gfCNCPoint5[10068] = {X 482.0421, Y 8.2448, Z -7.1667, A 0.000, B 0.000, C 0.000 }
gfCNCPoint5[10069] = {X 484.1469, Y 7.9173, Z -7.1667, A 0.000, B 0.000, C 0.000 }
gfCNCPoint5[10070] = {X 486.2738, Y 7.8018, Z -7.1667, A 0.000, B 0.000, C 0.000 }
gfCNCPoint5[10071] = {X 486.9707, Y 7.7896, Z -7.1667, A 0.000, B 0.000, C 0.000 }
gfCNCPoint5[10072] = {X 502.2084, Y 7.7896, Z -7.1667, A 0.000, B 0.000, C 0.000 }
gfCNCPoint5[10073] = {X 502.7401, Y 7.7937, Z -7.1667, A 0.000, B 0.000, C 0.000 }
gfCNCPoint5[10074] = {X 503.7097, Y 7.9101, Z -7.1667, A 0.000, B 0.000, C 0.000 }
gfCNCPoint5[10075] = {X 504.6294, Y 8.2383, Z -7.1667, A 0.000, B 0.000, C 0.000 }
gfCNCPoint5[10076] = {X 505.4537, Y 8.7620, Z -7.1667, A 0.000, B 0.000, C 0.000 }
gfCNCPoint5[10077] = {X 506.1415, Y 9.4552, Z -7.1667, A 0.000, B 0.000, C 0.000 }
gfCNCPoint5[10078] = {X 506.6587, Y 10.2835, Z -7.1667, A 0.000, B 0.000, C 0.000 }
gfCNCPoint5[10079] = {X 506.9797, Y 11.2058, Z -7.1667, A 0.000, B 0.000, C 0.000 }
gfCNCPoint5[10080] = {X 507.0885, Y 12.1762, Z -7.1667, A 0.000, B 0.000, C 0.000 }
gfCNCPoint5[10081] = {X 507.0883, Y 13.0233, Z -7.1667, A 0.000, B 0.000, C 0.000 }
gfCNCPoint5[10082] = {X 506.9800, Y 13.9491, Z -7.1667, A 0.000, B 0.000, C 0.000 }
gfCNCPoint5[10083] = {X 506.6792, Y 14.8313, Z -7.1667, A 0.000, B 0.000, C 0.000 }
gfCNCPoint5[10084] = {X 506.1993, Y 15.6303, Z -7.1667, A 0.000, B 0.000, C 0.000 }
gfCNCPoint5[10085] = {X 505.5618, Y 16.3103, Z -7.1667, A 0.000, B 0.000, C 0.000 }
gfCNCPoint5[10086] = {X 505.5621, Y 40.8767, Z -7.1667, A 0.000, B 0.000, C 0.000 }
gfCNCPoint5[10087] = {X 506.2062, Y 41.5658, Z -7.1667, A 0.000, B 0.000, C 0.000 }
gfCNCPoint5[10088] = {X 506.6887, Y 42.3763, Z -7.1667, A 0.000, B 0.000, C 0.000 }
gfCNCPoint5[10089] = {X 506.9874, Y 43.2710, Z -7.1667, A 0.000, B 0.000, C 0.000 }
gfCNCPoint5[10090] = {X 507.0885, Y 44.2089, Z -7.1667, A 0.000, B 0.000, C 0.000 }
gfCNCPoint5[10091] = {X 507.0885, Y 45.0000, Z -7.1667, A 0.000, B 0.000, C 0.000 }
gfCNCPoint5[10092] = {X 506.9782, Y 45.9791, Z -7.1667, A 0.000, B 0.000, C 0.000 }
gfCNCPoint5[10093] = {X 506.6528, Y 46.9091, Z -7.1667, A 0.000, B 0.000, C 0.000 }
gfCNCPoint5[10094] = {X 506.1285, Y 47.7434, Z -7.1667, A 0.000, B 0.000, C 0.000 }
gfCNCPoint5[10095] = {X 505.4318, Y 48.4401, Z -7.1667, A 0.000, B 0.000, C 0.000 }
gfCNCPoint5[10096] = {X 504.5976, Y 48.9643, Z -7.1667, A 0.000, B 0.000, C 0.000 }
gfCNCPoint5[10097] = {X 503.6676, Y 49.2897, Z -7.1667, A 0.000, B 0.000, C 0.000 }
gfCNCPoint5[10098] = {X 502.6885, Y 49.4000, Z -7.1667, A 0.000, B 0.000, C 0.000 }
gfCNCPoint5[10099] = {X 496.2450, Y 49.4000, Z -7.1667, A 0.000, B 0.000, C 0.000 }
gfCNCPoint5[10100] = {X 495.2659, Y 49.2897, Z -7.1667, A 0.000, B 0.000, C 0.000 }
gfCNCPoint5[10101] = {X 494.3359, Y 48.9643, Z -7.1667, A 0.000, B 0.000, C 0.000 }
gfCNCPoint5[10102] = {X 493.5017, Y 48.4401, Z -7.1667, A 0.000, B 0.000, C 0.000 }
gfCNCPoint5[10103] = {X 492.8050, Y 47.7433, Z -7.1667, A 0.000, B 0.000, C 0.000 }
gfCNCPoint5[10104] = {X 492.2808, Y 46.9091, Z -7.1667, A 0.000, B 0.000, C 0.000 }
gfCNCPoint5[10105] = {X 491.9553, Y 45.9791, Z -7.1667, A 0.000, B 0.000, C 0.000 }
gfCNCPoint5[10106] = {X 491.8450, Y 45.0000, Z -7.1667, A 0.000, B 0.000, C 0.000 }
gfCNCPoint5[10107] = {X 491.8454, Y 44.1483, Z -7.1667, A 0.000, B 0.000, C 0.000 }
gfCNCPoint5[10108] = {X 491.9559, Y 43.2275, Z -7.1667, A 0.000, B 0.000, C 0.000 }
gfCNCPoint5[10109] = {X 492.2568, Y 42.3503, Z -7.1667, A 0.000, B 0.000, C 0.000 }
gfCNCPoint5[10110] = {X 492.7349, Y 41.5556, Z -7.1667, A 0.000, B 0.000, C 0.000 }
gfCNCPoint5[10111] = {X 493.3690, Y 40.8789, Z -7.1667, A 0.000, B 0.000, C 0.000 }
gfCNCPoint5[10112] = {X 493.3690, Y 34.5538, Z -7.1667, A 0.000, B 0.000, C 0.000 }
gfCNCPoint5[10113] = {X 490.7743, Y 34.5538, Z -7.1667, A 0.000, B 0.000, C 0.000 }
gfCNCPoint5[10114] = {X 486.5274, Y 42.8240, Z -7.1667, A 0.000, B 0.000, C 0.000 }
gfCNCPoint5[10115] = {X 486.6948, Y 43.5075, Z -7.1667, A 0.000, B 0.000, C 0.000 }
gfCNCPoint5[10116] = {X 486.7510, Y 44.2089, Z -7.1667, A 0.000, B 0.000, C 0.000 }
gfCNCPoint5[10117] = {X 486.7510, Y 45.0000, Z -7.1667, A 0.000, B 0.000, C 0.000 }
gfCNCPoint5[10118] = {X 486.6407, Y 45.9791, Z -7.1667, A 0.000, B 0.000, C 0.000 }
gfCNCPoint5[10119] = {X 486.3153, Y 46.9091, Z -7.1667, A 0.000, B 0.000, C 0.000 }
gfCNCPoint5[10120] = {X 485.7911, Y 47.7434, Z -7.1667, A 0.000, B 0.000, C 0.000 }
gfCNCPoint5[10121] = {X 485.0944, Y 48.4401, Z -7.1667, A 0.000, B 0.000, C 0.000 }
gfCNCPoint5[10122] = {X 484.2601, Y 48.9643, Z -7.1667, A 0.000, B 0.000, C 0.000 }
gfCNCPoint5[10123] = {X 483.3301, Y 49.2897, Z -7.1667, A 0.000, B 0.000, C 0.000 }
gfCNCPoint5[10124] = {X 482.3510, Y 49.4000, Z -7.1667, A 0.000, B 0.000, C 0.000 }
gfCNCPoint5[10125] = {X 480.2695, Y 49.4000, Z -7.1667, A 0.000, B 0.000, C 0.000 }
gfCNCPoint5[10126] = {X 480.2695, Y 49.8800, Z -7.1667, A 0.000, B 0.000, C 0.000 }
gfCNCPoint5[10127] = {X 481.4067, Y 50.7435, Z -7.1667, A 0.000, B 0.000, C 0.000 }
gfCNCPoint5[10128] = {X 482.4044, Y 51.7649, Z -7.1667, A 0.000, B 0.000, C 0.000 }
gfCNCPoint5[10129] = {X 483.2411, Y 52.9219, Z -7.1667, A 0.000, B 0.000, C 0.000 }
gfCNCPoint5[10130] = {X 483.8615, Y 54.1044, Z -7.1667, A 0.000, B 0.000, C 0.000 }
gfCNCPoint5[10131] = {X 484.3133, Y 55.3610, Z -7.1667, A 0.000, B 0.000, C 0.000 }
gfCNCPoint5[10132] = {X 484.5879, Y 56.6678, Z -7.1667, A 0.000, B 0.000, C 0.000 }
gfCNCPoint5[10133] = {X 484.6800, Y 58.0000, Z -7.1667, A 0.000, B 0.000, C 0.000 }
gfCNCPoint5[10134] = {X 484.6797, Y 59.0140, Z -7.1667, A 0.000, B 0.000, C 0.000 }
gfCNCPoint5[10135] = {X 484.5592, Y 60.4583, Z -7.1667, A 0.000, B 0.000, C 0.000 }
gfCNCPoint5[10136] = {X 484.2246, Y 61.8683, Z -7.1667, A 0.000, B 0.000, C 0.000 }
gfCNCPoint5[10137] = {X 483.6831, Y 63.2126, Z -7.1667, A 0.000, B 0.000, C 0.000 }
gfCNCPoint5[10138] = {X 482.9471, Y 64.4610, Z -7.1667, A 0.000, B 0.000, C 0.000 }
gfCNCPoint5[10139] = {X 482.0329, Y 65.5855, Z -7.1667, A 0.000, B 0.000, C 0.000 }
gfCNCPoint5[10140] = {X 480.9610, Y 66.5609, Z -7.1667, A 0.000, B 0.000, C 0.000 }
gfCNCPoint5[10141] = {X 480.9614, Y 89.4451, Z -7.1667, A 0.000, B 0.000, C 0.000 }
gfCNCPoint5[10142] = {X 482.0603, Y 90.4475, Z -7.1667, A 0.000, B 0.000, C 0.000 }
gfCNCPoint5[10143] = {X 482.9923, Y 91.6066, Z -7.1667, A 0.000, B 0.000, C 0.000 }
gfCNCPoint5[10144] = {X 483.7353, Y 92.8951, Z -7.1667, A 0.000, B 0.000, C 0.000 }
gfCNCPoint5[10145] = {X 507.6812, Y 92.8951, Z -7.1667, A 0.000, B 0.000, C 0.000 }
gfCNCPoint5[10146] = {X 507.6812, Y 95.2951, Z -7.1667, A 0.000, B 0.000, C 0.000 }
gfCNCPoint5[10147] = {X 595.2967, Y 95.2951, Z -7.1667, A 0.000, B 0.000, C 0.000 }
gfCNCPoint5[10148] = {X 595.2967, Y 54.2000, Z -7.1667, A 0.000, B 0.000, C 0.000 }
gfCNCPoint5[10149] = {X 593.5565, Y 54.2000, Z -7.1667, A 0.000, B 0.000, C 0.000 }
gfCNCPoint5[10150] = {X 592.2403, Y 54.1053, Z -7.1667, A 0.000, B 0.000, C 0.000 }
gfCNCPoint5[10151] = {X 590.9511, Y 53.8233, Z -7.1667, A 0.000, B 0.000, C 0.000 }
gfCNCPoint5[10152] = {X 589.7155, Y 53.3598, Z -7.1667, A 0.000, B 0.000, C 0.000 }
gfCNCPoint5[10153] = {X 588.5589, Y 52.7242, Z -7.1667, A 0.000, B 0.000, C 0.000 }
gfCNCPoint5[10154] = {X 587.5052, Y 51.9297, Z -7.1667, A 0.000, B 0.000, C 0.000 }
gfCNCPoint5[10155] = {X 586.4956, Y 52.6955, Z -7.1667, A 0.000, B 0.000, C 0.000 }
gfCNCPoint5[10156] = {X 585.3903, Y 53.3153, Z -7.1667, A 0.000, B 0.000, C 0.000 }
gfCNCPoint5[10157] = {X 584.1375, Y 53.7999, Z -7.1667, A 0.000, B 0.000, C 0.000 }
gfCNCPoint5[10158] = {X 582.8276, Y 54.0969, Z -7.1667, A 0.000, B 0.000, C 0.000 }
gfCNCPoint5[10159] = {X 581.4884, Y 54.1999, Z -7.1667, A 0.000, B 0.000, C 0.000 }
gfCNCPoint5[10160] = {X 580.1485, Y 54.1069, Z -7.1667, A 0.000, B 0.000, C 0.000 }
gfCNCPoint5[10161] = {X 578.8364, Y 53.8198, Z -7.1667, A 0.000, B 0.000, C 0.000 }
gfCNCPoint5[10162] = {X 577.5801, Y 53.3447, Z -7.1667, A 0.000, B 0.000, C 0.000 }
gfCNCPoint5[10163] = {X 576.4063, Y 52.6917, Z -7.1667, A 0.000, B 0.000, C 0.000 }
gfCNCPoint5[10164] = {X 575.3401, Y 51.8748, Z -7.1667, A 0.000, B 0.000, C 0.000 }
gfCNCPoint5[10165] = {X 574.2798, Y 52.6879, Z -7.1667, A 0.000, B 0.000, C 0.000 }
gfCNCPoint5[10166] = {X 573.1128, Y 53.3388, Z -7.1667, A 0.000, B 0.000, C 0.000 }
gfCNCPoint5[10167] = {X 571.8638, Y 53.8139, Z -7.1667, A 0.000, B 0.000, C 0.000 }
gfCNCPoint5[10168] = {X 570.5592, Y 54.1030, Z -7.1667, A 0.000, B 0.000, C 0.000 }
gfCNCPoint5[10169] = {X 569.2264, Y 54.2000, Z -7.1667, A 0.000, B 0.000, C 0.000 }
gfCNCPoint5[10170] = {X 562.4443, Y 54.2000, Z -7.1667, A 0.000, B 0.000, C 0.000 }
gfCNCPoint5[10171] = {X 561.0051, Y 54.0867, Z -7.1667, A 0.000, B 0.000, C 0.000 }
gfCNCPoint5[10172] = {X 559.6013, Y 53.7497, Z -7.1667, A 0.000, B 0.000, C 0.000 }
gfCNCPoint5[10173] = {X 558.2676, Y 53.1973, Z -7.1667, A 0.000, B 0.000, C 0.000 }
gfCNCPoint5[10174] = {X 557.0367, Y 52.4430, Z -7.1667, A 0.000, B 0.000, C 0.000 }
gfCNCPoint5[10175] = {X 555.9389, Y 51.5054, Z -7.1667, A 0.000, B 0.000, C 0.000 }
gfCNCPoint5[10176] = {X 555.0013, Y 50.4076, Z -7.1667, A 0.000, B 0.000, C 0.000 }
gfCNCPoint5[10177] = {X 554.2470, Y 49.1767, Z -7.1667, A 0.000, B 0.000, C 0.000 }
gfCNCPoint5[10178] = {X 553.6946, Y 47.8430, Z -7.1667, A 0.000, B 0.000, C 0.000 }
gfCNCPoint5[10179] = {X 553.3576, Y 46.4392, Z -7.1667, A 0.000, B 0.000, C 0.000 }
gfCNCPoint5[10180] = {X 553.2443, Y 45.0000, Z -7.1667, A 0.000, B 0.000, C 0.000 }
gfCNCPoint5[10181] = {X 553.2443, Y 44.0484, Z -7.1667, A 0.000, B 0.000, C 0.000 }
gfCNCPoint5[10182] = {X 553.3457, Y 42.7151, Z -7.1667, A 0.000, B 0.000, C 0.000 }
gfCNCPoint5[10183] = {X 553.6387, Y 41.4104, Z -7.1667, A 0.000, B 0.000, C 0.000 }
gfCNCPoint5[10184] = {X 554.1171, Y 40.1617, Z -7.1667, A 0.000, B 0.000, C 0.000 }
gfCNCPoint5[10185] = {X 554.7709, Y 38.9953, Z -7.1667, A 0.000, B 0.000, C 0.000 }
gfCNCPoint5[10186] = {X 554.7710, Y 11.0096, Z -7.1667, A 0.000, B 0.000, C 0.000 }
gfCNCPoint5[10187] = {X 554.1214, Y 9.8543, Z -7.1667, A 0.000, B 0.000, C 0.000 }
gfCNCPoint5[10188] = {X 553.6444, Y 8.6178, Z -7.1667, A 0.000, B 0.000, C 0.000 }
gfCNCPoint5[10189] = {X 553.3501, Y 7.3255, Z -7.1667, A 0.000, B 0.000, C 0.000 }
gfCNCPoint5[10190] = {X 553.2446, Y 6.0043, Z -7.1667, A 0.000, B 0.000, C 0.000 }
gfCNCPoint5[10191] = {X 553.2443, Y 5.0000, Z -7.1667, A 0.000, B 0.000, C 0.000 }
gfCNCPoint5[10192] = {X 553.2455, Y 4.8524, Z -7.1667, A 0.000, B 0.000, C 0.000 }
gfCNCPoint5[10193] = {X 553.2490, Y 4.7049, Z -7.1667, A 0.000, B 0.000, C 0.000 }
gfCNCPoint5[10194] = {X 365.1895, Y 4.7049, Z -7.1667, A 0.000, B 0.000, C 0.000 }
gfCNCPoint5[10195] = {X 365.3287, Y 4.8540, Z -7.1667, A 0.000, B 0.000, C 0.000 }
gfCNCPoint5[10196] = {X 366.7808, Y 6.5792, Z -7.1667, A 0.000, B 0.000, C 0.000 }
gfCNCPoint5[10197] = {X 368.0884, Y 8.4162, Z -7.1667, A 0.000, B 0.000, C 0.000 }
gfCNCPoint5[10198] = {X 369.2513, Y 10.3687, Z -7.1667, A 0.000, B 0.000, C 0.000 }
gfCNCPoint5[10199] = {X 370.2509, Y 12.4095, Z -7.1667, A 0.000, B 0.000, C 0.000 }
gfCNCPoint5[10200] = {X 371.0806, Y 14.5252, Z -7.1667, A 0.000, B 0.000, C 0.000 }
gfCNCPoint5[10201] = {X 371.7348, Y 16.7015, Z -7.1667, A 0.000, B 0.000, C 0.000 }
gfCNCPoint5[10202] = {X 372.2634, Y 19.2108, Z -7.1667, A 0.000, B 0.000, C 0.000 }
gfCNCPoint5[10203] = {X 372.6044, Y 21.7523, Z -7.1667, A 0.000, B 0.000, C 0.000 }
gfCNCPoint5[10204] = {X 372.7559, Y 24.3122, Z -7.1667, A 0.000, B 0.000, C 0.000 }
gfCNCPoint5[10205] = {X 372.7172, Y 26.8762, Z -7.1667, A 0.000, B 0.000, C 0.000 }
gfCNCPoint5[10206] = {X 372.4884, Y 29.4303, Z -7.1667, A 0.000, B 0.000, C 0.000 }
gfCNCPoint5[10207] = {X 372.0708, Y 31.9604, Z -7.1667, A 0.000, B 0.000, C 0.000 }
gfCNCPoint5[10208] = {X 371.4839, Y 34.3164, Z -7.1667, A 0.000, B 0.000, C 0.000 }
gfCNCPoint5[10209] = {X 370.6915, Y 36.6115, Z -7.1667, A 0.000, B 0.000, C 0.000 }
gfCNCPoint5[10210] = {X 369.6997, Y 38.8278, Z -7.1667, A 0.000, B 0.000, C 0.000 }
gfCNCPoint5[10211] = {X 368.5162, Y 40.9478, Z -7.1667, A 0.000, B 0.000, C 0.000 }
gfCNCPoint5[10212] = {X 367.1503, Y 42.9553, Z -7.1667, A 0.000, B 0.000, C 0.000 }
gfCNCPoint5[10213] = {X 365.8289, Y 44.5915, Z -7.1667, A 0.000, B 0.000, C 0.000 }
gfCNCPoint5[10214] = {X 364.3743, Y 46.1106, Z -7.1667, A 0.000, B 0.000, C 0.000 }
gfCNCPoint5[10215] = {X 362.7970, Y 47.5018, Z -7.1667, A 0.000, B 0.000, C 0.000 }
gfCNCPoint5[10216] = {X 361.1080, Y 48.7552, Z -7.1667, A 0.000, B 0.000, C 0.000 }
gfCNCPoint5[10217] = {X 359.3195, Y 49.8618, Z -7.1667, A 0.000, B 0.000, C 0.000 }
gfCNCPoint5[10218] = {X 357.4441, Y 50.8138, Z -7.1667, A 0.000, B 0.000, C 0.000 }
gfCNCPoint5[10219] = {X 355.4664, Y 51.5796, Z -7.1667, A 0.000, B 0.000, C 0.000 }
gfCNCPoint5[10220] = {X 353.4327, Y 52.1816, Z -7.1667, A 0.000, B 0.000, C 0.000 }
gfCNCPoint5[10221] = {X 351.3568, Y 52.6157, Z -7.1667, A 0.000, B 0.000, C 0.000 }
gfCNCPoint5[10222] = {X 349.2523, Y 52.8790, Z -7.1667, A 0.000, B 0.000, C 0.000 }
gfCNCPoint5[10223] = {X 347.1334, Y 52.9699, Z -7.1667, A 0.000, B 0.000, C 0.000 }
gfCNCPoint5[10224] = {X 344.8131, Y 52.9275, Z -7.1667, A 0.000, B 0.000, C 0.000 }
gfCNCPoint5[10225] = {X 342.5052, Y 52.6844, Z -7.1667, A 0.000, B 0.000, C 0.000 }
gfCNCPoint5[10226] = {X 340.2270, Y 52.2423, Z -7.1667, A 0.000, B 0.000, C 0.000 }
gfCNCPoint5[10227] = {X 337.9956, Y 51.6045, Z -7.1667, A 0.000, B 0.000, C 0.000 }
gfCNCPoint5[10228] = {X 335.8279, Y 50.7758, Z -7.1667, A 0.000, B 0.000, C 0.000 }
gfCNCPoint5[10229] = {X 333.7401, Y 49.7625, Z -7.1667, A 0.000, B 0.000, C 0.000 }
gfCNCPoint5[10230] = {X 332.8361, Y 49.2300, Z -7.1667, A 0.000, B 0.000, C 0.000 }
gfCNCPoint5[10231] = {X 331.9535, Y 48.6626, Z -7.1667, A 0.000, B 0.000, C 0.000 }
gfCNCPoint5[10232] = {X 331.3040, Y 48.2128, Z -7.1667, A 0.000, B 0.000, C 0.000 }
gfCNCPoint5[10233] = {X 330.6681, Y 47.7441, Z -7.1667, A 0.000, B 0.000, C 0.000 }
gfCNCPoint5[10234] = {X 329.2159, Y 49.6549, Z -7.1667, A 0.000, B 0.000, C 0.000 }
gfCNCPoint5[10235] = {X 328.8717, Y 49.3893, Z -7.1667, A 0.000, B 0.000, C 0.000 }
gfCNCPoint5[10236] = {X 328.5316, Y 49.1185, Z -7.1667, A 0.000, B 0.000, C 0.000 }
gfCNCPoint5[10237] = {X 328.1266, Y 49.0390, Z -7.1667, A 0.000, B 0.000, C 0.000 }
gfCNCPoint5[10238] = {X 327.7253, Y 48.9423, Z -7.1667, A 0.000, B 0.000, C 0.000 }
gfCNCPoint5[10239] = {X 328.4858, Y 49.2667, Z -7.1667, A 0.000, B 0.000, C 0.000 }
gfCNCPoint5[10240] = {X 329.2159, Y 49.6549, Z -7.1667, A 0.000, B 0.000, C 0.000 }
gfCNCPoint5[10241] = {X 330.6681, Y 47.7441, Z -7.1667, A 0.000, B 0.000, C 0.000 }
gfCNCPoint5[10242] = {X 330.0947, Y 47.2959, Z -7.1667, A 0.000, B 0.000, C 0.000 }
gfCNCPoint5[10243] = {X 329.5337, Y 46.8324, Z -7.1667, A 0.000, B 0.000, C 0.000 }
gfCNCPoint5[10244] = {X 328.9312, Y 46.7520, Z -7.1667, A 0.000, B 0.000, C 0.000 }
gfCNCPoint5[10245] = {X 328.3374, Y 46.6216, Z -7.1667, A 0.000, B 0.000, C 0.000 }
gfCNCPoint5[10246] = {X 327.9789, Y 46.5172, Z -7.1667, A 0.000, B 0.000, C 0.000 }
gfCNCPoint5[10247] = {X 327.6263, Y 46.3944, Z -7.1667, A 0.000, B 0.000, C 0.000 }
gfCNCPoint5[10248] = {X 326.7320, Y 45.9864, Z -7.1667, A 0.000, B 0.000, C 0.000 }
gfCNCPoint5[10249] = {X 325.9009, Y 45.4616, Z -7.1667, A 0.000, B 0.000, C 0.000 }
gfCNCPoint5[10250] = {X 325.1480, Y 44.8296, Z -7.1667, A 0.000, B 0.000, C 0.000 }
gfCNCPoint5[10251] = {X 324.5140, Y 44.2115, Z -7.1667, A 0.000, B 0.000, C 0.000 }
gfCNCPoint5[10252] = {X 324.0475, Y 43.7117, Z -7.1667, A 0.000, B 0.000, C 0.000 }
gfCNCPoint5[10253] = {X 323.6300, Y 43.1703, Z -7.1667, A 0.000, B 0.000, C 0.000 }
gfCNCPoint5[10254] = {X 319.6957, Y 45.9200, Z -7.1667, A 0.000, B 0.000, C 0.000 }
gfCNCPoint5[10255] = {X 319.4780, Y 45.5976, Z -7.1667, A 0.000, B 0.000, C 0.000 }
gfCNCPoint5[10256] = {X 319.2708, Y 45.2683, Z -7.1667, A 0.000, B 0.000, C 0.000 }
gfCNCPoint5[10257] = {X 319.2514, Y 45.5948, Z -7.1667, A 0.000, B 0.000, C 0.000 }
gfCNCPoint5[10258] = {X 319.2174, Y 45.9200, Z -7.1667, A 0.000, B 0.000, C 0.000 }
gfCNCPoint5[10259] = {X 319.6957, Y 45.9200, Z -7.1667, A 0.000, B 0.000, C 0.000 }
gfCNCPoint5[10260] = {X 321.6628, Y 44.5452, Z -7.1667, A 0.000, B 0.000, C 0.000 }
gfCNCPoint5[10261] = {X 321.4884, Y 44.2868, Z -7.1667, A 0.000, B 0.000, C 0.000 }
gfCNCPoint5[10262] = {X 321.3224, Y 44.0230, Z -7.1667, A 0.000, B 0.000, C 0.000 }
gfCNCPoint5[10263] = {X 320.6708, Y 42.7446, Z -7.1667, A 0.000, B 0.000, C 0.000 }
gfCNCPoint5[10264] = {X 320.2153, Y 41.3839, Z -7.1667, A 0.000, B 0.000, C 0.000 }
gfCNCPoint5[10265] = {X 319.9660, Y 39.9709, Z -7.1667, A 0.000, B 0.000, C 0.000 }
gfCNCPoint5[10266] = {X 319.9283, Y 38.5365, Z -7.1667, A 0.000, B 0.000, C 0.000 }
gfCNCPoint5[10267] = {X 320.1030, Y 37.1123, Z -7.1667, A 0.000, B 0.000, C 0.000 }
gfCNCPoint5[10268] = {X 320.4312, Y 35.8877, Z -7.1667, A 0.000, B 0.000, C 0.000 }
gfCNCPoint5[10269] = {X 320.9165, Y 34.7164, Z -7.1667, A 0.000, B 0.000, C 0.000 }
gfCNCPoint5[10270] = {X 321.5508, Y 33.6186, Z -7.1667, A 0.000, B 0.000, C 0.000 }
gfCNCPoint5[10271] = {X 324.1392, Y 29.7485, Z -7.1667, A 0.000, B 0.000, C 0.000 }
gfCNCPoint5[10272] = {X 320.1493, Y 27.0800, Z -7.1667, A 0.000, B 0.000, C 0.000 }
gfCNCPoint5[10273] = {X 321.8041, Y 24.6057, Z -7.1667, A 0.000, B 0.000, C 0.000 }
gfCNCPoint5[10274] = {X 321.9897, Y 24.3356, Z -7.1667, A 0.000, B 0.000, C 0.000 }
gfCNCPoint5[10275] = {X 322.1814, Y 24.0697, Z -7.1667, A 0.000, B 0.000, C 0.000 }
gfCNCPoint5[10276] = {X 321.5380, Y 23.0772, Z -7.1667, A 0.000, B 0.000, C 0.000 }
gfCNCPoint5[10277] = {X 320.9777, Y 22.0354, Z -7.1667, A 0.000, B 0.000, C 0.000 }
gfCNCPoint5[10278] = {X 320.1494, Y 20.3316, Z -7.1667, A 0.000, B 0.000, C 0.000 }
gfCNCPoint5[10279] = {X 320.1493, Y 27.0800, Z -7.1667, A 0.000, B 0.000, C 0.000 }
gfCNCPoint5[10280] = {X 322.1442, Y 28.4143, Z -7.1667, A 0.000, B 0.000, C 0.000 }
gfCNCPoint5[10281] = {X 323.7974, Y 25.9424, Z -7.1667, A 0.000, B 0.000, C 0.000 }
gfCNCPoint5[10282] = {X 324.5112, Y 24.9841, Z -7.1667, A 0.000, B 0.000, C 0.000 }
gfCNCPoint5[10283] = {X 325.3162, Y 24.1010, Z -7.1667, A 0.000, B 0.000, C 0.000 }
gfCNCPoint5[10284] = {X 324.4812, Y 23.1413, Z -7.1667, A 0.000, B 0.000, C 0.000 }
gfCNCPoint5[10285] = {X 323.7518, Y 22.0990, Z -7.1667, A 0.000, B 0.000, C 0.000 }
gfCNCPoint5[10286] = {X 323.1360, Y 20.9859, Z -7.1667, A 0.000, B 0.000, C 0.000 }
gfCNCPoint5[10287] = {X 319.6151, Y 13.7428, Z -7.1667, A 0.000, B 0.000, C 0.000 }
gfCNCPoint5[10288] = {X 319.4387, Y 13.3633, Z -7.1667, A 0.000, B 0.000, C 0.000 }
gfCNCPoint5[10289] = {X 319.2755, Y 12.9779, Z -7.1667, A 0.000, B 0.000, C 0.000 }
gfCNCPoint5[10290] = {X 319.2755, Y 13.0353, Z -7.1667, A 0.000, B 0.000, C 0.000 }
gfCNCPoint5[10291] = {X 319.1699, Y 14.2150, Z -7.1667, A 0.000, B 0.000, C 0.000 }
gfCNCPoint5[10292] = {X 318.8743, Y 15.3621, Z -7.1667, A 0.000, B 0.000, C 0.000 }
gfCNCPoint5[10293] = {X 318.3966, Y 16.4460, Z -7.1667, A 0.000, B 0.000, C 0.000 }
gfCNCPoint5[10294] = {X 317.7495, Y 17.4381, Z -7.1667, A 0.000, B 0.000, C 0.000 }
gfCNCPoint5[10295] = {X 317.7491, Y 36.6443, Z -7.1667, A 0.000, B 0.000, C 0.000 }
gfCNCPoint5[10296] = {X 318.1586, Y 35.1160, Z -7.1667, A 0.000, B 0.000, C 0.000 }
gfCNCPoint5[10297] = {X 318.7643, Y 33.6544, Z -7.1667, A 0.000, B 0.000, C 0.000 }
gfCNCPoint5[10298] = {X 319.5559, Y 32.2844, Z -7.1667, A 0.000, B 0.000, C 0.000 }
gfCNCPoint5[10299] = {X 322.1442, Y 28.4143, Z -7.1667, A 0.000, B 0.000, C 0.000 }
gfCNCPoint5[10300] = {X 324.1392, Y 29.7485, Z -7.1667, A 0.000, B 0.000, C 0.000 }
gfCNCPoint5[10301] = {X 325.7907, Y 27.2791, Z -7.1667, A 0.000, B 0.000, C 0.000 }
gfCNCPoint5[10302] = {X 326.3627, Y 26.5112, Z -7.1667, A 0.000, B 0.000, C 0.000 }
gfCNCPoint5[10303] = {X 327.0077, Y 25.8035, Z -7.1667, A 0.000, B 0.000, C 0.000 }
gfCNCPoint5[10304] = {X 328.0707, Y 24.8904, Z -7.1667, A 0.000, B 0.000, C 0.000 }
gfCNCPoint5[10305] = {X 329.2543, Y 24.1403, Z -7.1667, A 0.000, B 0.000, C 0.000 }
gfCNCPoint5[10306] = {X 328.0859, Y 23.3667, Z -7.1667, A 0.000, B 0.000, C 0.000 }
gfCNCPoint5[10307] = {X 327.0414, Y 22.4326, Z -7.1667, A 0.000, B 0.000, C 0.000 }
gfCNCPoint5[10308] = {X 326.3723, Y 21.6635, Z -7.1667, A 0.000, B 0.000, C 0.000 }
gfCNCPoint5[10309] = {X 325.7878, Y 20.8284, Z -7.1667, A 0.000, B 0.000, C 0.000 }
gfCNCPoint5[10310] = {X 325.2944, Y 19.9364, Z -7.1667, A 0.000, B 0.000, C 0.000 }
gfCNCPoint5[10311] = {X 321.7736, Y 12.6936, Z -7.1667, A 0.000, B 0.000, C 0.000 }
gfCNCPoint5[10312] = {X 321.6322, Y 12.3894, Z -7.1667, A 0.000, B 0.000, C 0.000 }
gfCNCPoint5[10313] = {X 321.5015, Y 12.0806, Z -7.1667, A 0.000, B 0.000, C 0.000 }
gfCNCPoint5[10314] = {X 321.1058, Y 10.8773, Z -7.1667, A 0.000, B 0.000, C 0.000 }
gfCNCPoint5[10315] = {X 320.8706, Y 9.6327, Z -7.1667, A 0.000, B 0.000, C 0.000 }
gfCNCPoint5[10316] = {X 320.7999, Y 8.3680, Z -7.1667, A 0.000, B 0.000, C 0.000 }
gfCNCPoint5[10317] = {X 320.8950, Y 7.1049, Z -7.1667, A 0.000, B 0.000, C 0.000 }
gfCNCPoint5[10318] = {X 298.7843, Y 7.1049, Z -7.1667, A 0.000, B 0.000, C 0.000 }
gfCNCPoint5[10319] = {X 298.7843, Y 9.5049, Z -7.1667, A 0.000, B 0.000, C 0.000 }
gfCNCPoint5[10320] = {X 297.8291, Y 9.5049, Z -7.1667, A 0.000, B 0.000, C 0.000 }
gfCNCPoint5[10321] = {X 298.1371, Y 10.4755, Z -7.1667, A 0.000, B 0.000, C 0.000 }
gfCNCPoint5[10322] = {X 298.3067, Y 11.4795, Z -7.1667, A 0.000, B 0.000, C 0.000 }
gfCNCPoint5[10323] = {X 298.4763, Y 10.4755, Z -7.1667, A 0.000, B 0.000, C 0.000 }
gfCNCPoint5[10324] = {X 298.7843, Y 9.5049, Z -7.1667, A 0.000, B 0.000, C 0.000 }
gfCNCPoint5[10325] = {X 298.7843, Y 7.1049, Z -7.1667, A 0.000, B 0.000, C 0.000 }
gfCNCPoint5[10326] = {X 191.0969, Y 7.1049, Z -7.1667, A 0.000, B 0.000, C 0.000 }
gfCNCPoint5[10327] = {X 193.0698, Y 7.6379, Z -7.1667, A 0.000, B 0.000, C 0.000 }
gfCNCPoint5[10328] = {X 194.9678, Y 8.3954, Z -7.1667, A 0.000, B 0.000, C 0.000 }
gfCNCPoint5[10329] = {X 196.7657, Y 9.3671, Z -7.1667, A 0.000, B 0.000, C 0.000 }
gfCNCPoint5[10330] = {X 198.4393, Y 10.5400, Z -7.1667, A 0.000, B 0.000, C 0.000 }
gfCNCPoint5[10331] = {X 198.8606, Y 10.8896, Z -7.1667, A 0.000, B 0.000, C 0.000 }
gfCNCPoint5[10332] = {X 199.2675, Y 11.2559, Z -7.1667, A 0.000, B 0.000, C 0.000 }
gfCNCPoint5[10333] = {X 200.3527, Y 12.3983, Z -7.1667, A 0.000, B 0.000, C 0.000 }
gfCNCPoint5[10334] = {X 201.2982, Y 13.6587, Z -7.1667, A 0.000, B 0.000, C 0.000 }
gfCNCPoint5[10335] = {X 202.0914, Y 15.0200, Z -7.1667, A 0.000, B 0.000, C 0.000 }
gfCNCPoint5[10336] = {X 202.7217, Y 16.4641, Z -7.1667, A 0.000, B 0.000, C 0.000 }
gfCNCPoint5[10337] = {X 203.2153, Y 18.1838, Z -7.1667, A 0.000, B 0.000, C 0.000 }
gfCNCPoint5[10338] = {X 203.5086, Y 19.9487, Z -7.1667, A 0.000, B 0.000, C 0.000 }
gfCNCPoint5[10339] = {X 203.5977, Y 21.7356, Z -7.1667, A 0.000, B 0.000, C 0.000 }
gfCNCPoint5[10340] = {X 203.4813, Y 23.5210, Z -7.1667, A 0.000, B 0.000, C 0.000 }
gfCNCPoint5[10341] = {X 203.1611, Y 25.2812, Z -7.1667, A 0.000, B 0.000, C 0.000 }
gfCNCPoint5[10342] = {X 202.7606, Y 26.6267, Z -7.1667, A 0.000, B 0.000, C 0.000 }
gfCNCPoint5[10343] = {X 202.2089, Y 27.9175, Z -7.1667, A 0.000, B 0.000, C 0.000 }
gfCNCPoint5[10344] = {X 201.5132, Y 29.1368, Z -7.1667, A 0.000, B 0.000, C 0.000 }
gfCNCPoint5[10345] = {X 200.6827, Y 30.2685, Z -7.1667, A 0.000, B 0.000, C 0.000 }
gfCNCPoint5[10346] = {X 199.7282, Y 31.2978, Z -7.1667, A 0.000, B 0.000, C 0.000 }
gfCNCPoint5[10347] = {X 200.5673, Y 31.8703, Z -7.1667, A 0.000, B 0.000, C 0.000 }
gfCNCPoint5[10348] = {X 201.2697, Y 32.6040, Z -7.1667, A 0.000, B 0.000, C 0.000 }
gfCNCPoint5[10349] = {X 201.8050, Y 33.4673, Z -7.1667, A 0.000, B 0.000, C 0.000 }
gfCNCPoint5[10350] = {X 204.8262, Y 39.7091, Z -7.1667, A 0.000, B 0.000, C 0.000 }
gfCNCPoint5[10351] = {X 205.1508, Y 40.5847, Z -7.1667, A 0.000, B 0.000, C 0.000 }
gfCNCPoint5[10352] = {X 205.3026, Y 41.5062, Z -7.1667, A 0.000, B 0.000, C 0.000 }
gfCNCPoint5[10353] = {X 205.2761, Y 42.4397, Z -7.1667, A 0.000, B 0.000, C 0.000 }
gfCNCPoint5[10354] = {X 205.0723, Y 43.3511, Z -7.1667, A 0.000, B 0.000, C 0.000 }
gfCNCPoint5[10355] = {X 204.6986, Y 44.2070, Z -7.1667, A 0.000, B 0.000, C 0.000 }
gfCNCPoint5[10356] = {X 204.1687, Y 44.9760, Z -7.1667, A 0.000, B 0.000, C 0.000 }
gfCNCPoint5[10357] = {X 203.5020, Y 45.6299, Z -7.1667, A 0.000, B 0.000, C 0.000 }
gfCNCPoint5[10358] = {X 202.9658, Y 46.0634, Z -7.1667, A 0.000, B 0.000, C 0.000 }
gfCNCPoint5[10359] = {X 202.2139, Y 46.5641, Z -7.1667, A 0.000, B 0.000, C 0.000 }
gfCNCPoint5[10360] = {X 201.3829, Y 46.9179, Z -7.1667, A 0.000, B 0.000, C 0.000 }
gfCNCPoint5[10361] = {X 200.5009, Y 47.1130, Z -7.1667, A 0.000, B 0.000, C 0.000 }
gfCNCPoint5[10362] = {X 199.5981, Y 47.1427, Z -7.1667, A 0.000, B 0.000, C 0.000 }
gfCNCPoint5[10363] = {X 198.7052, Y 47.0058, Z -7.1667, A 0.000, B 0.000, C 0.000 }
gfCNCPoint5[10364] = {X 196.6158, Y 48.0778, Z -7.1667, A 0.000, B 0.000, C 0.000 }
gfCNCPoint5[10365] = {X 194.4464, Y 48.9771, Z -7.1667, A 0.000, B 0.000, C 0.000 }
gfCNCPoint5[10366] = {X 192.2114, Y 49.6979, Z -7.1667, A 0.000, B 0.000, C 0.000 }
gfCNCPoint5[10367] = {X 190.6551, Y 50.0841, Z -7.1667, A 0.000, B 0.000, C 0.000 }
gfCNCPoint5[10368] = {X 189.0757, Y 50.3609, Z -7.1667, A 0.000, B 0.000, C 0.000 }
gfCNCPoint5[10369] = {X 186.8996, Y 50.5594, Z -7.1667, A 0.000, B 0.000, C 0.000 }
gfCNCPoint5[10370] = {X 184.7144, Y 50.5503, Z -7.1667, A 0.000, B 0.000, C 0.000 }
gfCNCPoint5[10371] = {X 184.7393, Y 50.0709, Z -7.1667, A 0.000, B 0.000, C 0.000 }
gfCNCPoint5[10372] = {X 182.7588, Y 49.8802, Z -7.1667, A 0.000, B 0.000, C 0.000 }
gfCNCPoint5[10373] = {X 180.8029, Y 49.5152, Z -7.1667, A 0.000, B 0.000, C 0.000 }
gfCNCPoint5[10374] = {X 178.9539, Y 48.9792, Z -7.1667, A 0.000, B 0.000, C 0.000 }
gfCNCPoint5[10375] = {X 177.1791, Y 48.2337, Z -7.1667, A 0.000, B 0.000, C 0.000 }
gfCNCPoint5[10376] = {X 175.5020, Y 47.2885, Z -7.1667, A 0.000, B 0.000, C 0.000 }
gfCNCPoint5[10377] = {X 173.9450, Y 46.1562, Z -7.1667, A 0.000, B 0.000, C 0.000 }
gfCNCPoint5[10378] = {X 172.7967, Y 45.1084, Z -7.1667, A 0.000, B 0.000, C 0.000 }
gfCNCPoint5[10379] = {X 171.7806, Y 43.9319, Z -7.1667, A 0.000, B 0.000, C 0.000 }
gfCNCPoint5[10380] = {X 170.9109, Y 42.6435, Z -7.1667, A 0.000, B 0.000, C 0.000 }
gfCNCPoint5[10381] = {X 170.1998, Y 41.2611, Z -7.1667, A 0.000, B 0.000, C 0.000 }
gfCNCPoint5[10382] = {X 169.6574, Y 39.8043, Z -7.1667, A 0.000, B 0.000, C 0.000 }
gfCNCPoint5[10383] = {X 169.2913, Y 38.2935, Z -7.1667, A 0.000, B 0.000, C 0.000 }
gfCNCPoint5[10384] = {X 169.1807, Y 37.5991, Z -7.1667, A 0.000, B 0.000, C 0.000 }
gfCNCPoint5[10385] = {X 169.0218, Y 35.9858, Z -7.1667, A 0.000, B 0.000, C 0.000 }
gfCNCPoint5[10386] = {X 169.0391, Y 34.3647, Z -7.1667, A 0.000, B 0.000, C 0.000 }
gfCNCPoint5[10387] = {X 169.2323, Y 32.7552, Z -7.1667, A 0.000, B 0.000, C 0.000 }
gfCNCPoint5[10388] = {X 169.5992, Y 31.1761, Z -7.1667, A 0.000, B 0.000, C 0.000 }
gfCNCPoint5[10389] = {X 170.1355, Y 29.6463, Z -7.1667, A 0.000, B 0.000, C 0.000 }
gfCNCPoint5[10390] = {X 170.7622, Y 28.3586, Z -7.1667, A 0.000, B 0.000, C 0.000 }
gfCNCPoint5[10391] = {X 171.5519, Y 27.1640, Z -7.1667, A 0.000, B 0.000, C 0.000 }
gfCNCPoint5[10392] = {X 172.4910, Y 26.0828, Z -7.1667, A 0.000, B 0.000, C 0.000 }
gfCNCPoint5[10393] = {X 173.5633, Y 25.1336, Z -7.1667, A 0.000, B 0.000, C 0.000 }
gfCNCPoint5[10394] = {X 174.7504, Y 24.3327, Z -7.1667, A 0.000, B 0.000, C 0.000 }
gfCNCPoint5[10395] = {X 173.9906, Y 23.9224, Z -7.1667, A 0.000, B 0.000, C 0.000 }
gfCNCPoint5[10396] = {X 173.3256, Y 23.3716, Z -7.1667, A 0.000, B 0.000, C 0.000 }
gfCNCPoint5[10397] = {X 172.7809, Y 22.7014, Z -7.1667, A 0.000, B 0.000, C 0.000 }
gfCNCPoint5[10398] = {X 172.3776, Y 21.9378, Z -7.1667, A 0.000, B 0.000, C 0.000 }
gfCNCPoint5[10399] = {X 169.7664, Y 15.5423, Z -7.1667, A 0.000, B 0.000, C 0.000 }
gfCNCPoint5[10400] = {X 169.5125, Y 14.6752, Z -7.1667, A 0.000, B 0.000, C 0.000 }
gfCNCPoint5[10401] = {X 169.4412, Y 13.7745, Z -7.1667, A 0.000, B 0.000, C 0.000 }
gfCNCPoint5[10402] = {X 169.5553, Y 12.8782, Z -7.1667, A 0.000, B 0.000, C 0.000 }
gfCNCPoint5[10403] = {X 169.8501, Y 12.0241, Z -7.1667, A 0.000, B 0.000, C 0.000 }
gfCNCPoint5[10404] = {X 170.3131, Y 11.2482, Z -7.1667, A 0.000, B 0.000, C 0.000 }
gfCNCPoint5[10405] = {X 170.9249, Y 10.5833, Z -7.1667, A 0.000, B 0.000, C 0.000 }
gfCNCPoint5[10406] = {X 171.6596, Y 10.0573, Z -7.1667, A 0.000, B 0.000, C 0.000 }
gfCNCPoint5[10407] = {X 172.2916, Y 9.6970, Z -7.1667, A 0.000, B 0.000, C 0.000 }
gfCNCPoint5[10408] = {X 173.1773, Y 9.3227, Z -7.1667, A 0.000, B 0.000, C 0.000 }
gfCNCPoint5[10409] = {X 174.1231, Y 9.1497, Z -7.1667, A 0.000, B 0.000, C 0.000 }
gfCNCPoint5[10410] = {X 175.0839, Y 9.1863, Z -7.1667, A 0.000, B 0.000, C 0.000 }
gfCNCPoint5[10411] = {X 176.0139, Y 9.4307, Z -7.1667, A 0.000, B 0.000, C 0.000 }
gfCNCPoint5[10412] = {X 177.0965, Y 8.9703, Z -7.1667, A 0.000, B 0.000, C 0.000 }
gfCNCPoint5[10413] = {X 179.2738, Y 8.1689, Z -7.1667, A 0.000, B 0.000, C 0.000 }
gfCNCPoint5[10414] = {X 181.5196, Y 7.5862, Z -7.1667, A 0.000, B 0.000, C 0.000 }
gfCNCPoint5[10415] = {X 183.8118, Y 7.2279, Z -7.1667, A 0.000, B 0.000, C 0.000 }
gfCNCPoint5[10416] = {X 186.1283, Y 7.0975, Z -7.1667, A 0.000, B 0.000, C 0.000 }
gfCNCPoint5[10417] = {X 188.4463, Y 7.1963, Z -7.1667, A 0.000, B 0.000, C 0.000 }
gfCNCPoint5[10418] = {X 190.7432, Y 7.5234, Z -7.1667, A 0.000, B 0.000, C 0.000 }
gfCNCPoint5[10419] = {X 192.3398, Y 7.9118, Z -7.1667, A 0.000, B 0.000, C 0.000 }
gfCNCPoint5[10420] = {X 193.8919, Y 8.4510, Z -7.1667, A 0.000, B 0.000, C 0.000 }
gfCNCPoint5[10421] = {X 195.3854, Y 9.1361, Z -7.1667, A 0.000, B 0.000, C 0.000 }
gfCNCPoint5[10422] = {X 196.8066, Y 9.9607, Z -7.1667, A 0.000, B 0.000, C 0.000 }
gfCNCPoint5[10423] = {X 198.1426, Y 10.9173, Z -7.1667, A 0.000, B 0.000, C 0.000 }
gfCNCPoint5[10424] = {X 199.2094, Y 11.8667, Z -7.1667, A 0.000, B 0.000, C 0.000 }
gfCNCPoint5[10425] = {X 200.1665, Y 12.9264, Z -7.1667, A 0.000, B 0.000, C 0.000 }
gfCNCPoint5[10426] = {X 201.0026, Y 14.0840, Z -7.1667, A 0.000, B 0.000, C 0.000 }
gfCNCPoint5[10427] = {X 201.7078, Y 15.3258, Z -7.1667, A 0.000, B 0.000, C 0.000 }
gfCNCPoint5[10428] = {X 202.2737, Y 16.6369, Z -7.1667, A 0.000, B 0.000, C 0.000 }
gfCNCPoint5[10429] = {X 202.7499, Y 18.3014, Z -7.1667, A 0.000, B 0.000, C 0.000 }
gfCNCPoint5[10430] = {X 203.0325, Y 20.0095, Z -7.1667, A 0.000, B 0.000, C 0.000 }
gfCNCPoint5[10431] = {X 203.1177, Y 21.7387, Z -7.1667, A 0.000, B 0.000, C 0.000 }
gfCNCPoint5[10432] = {X 203.0045, Y 23.4663, Z -7.1667, A 0.000, B 0.000, C 0.000 }
gfCNCPoint5[10433] = {X 202.6943, Y 25.1696, Z -7.1667, A 0.000, B 0.000, C 0.000 }
gfCNCPoint5[10434] = {X 202.2595, Y 26.5986, Z -7.1667, A 0.000, B 0.000, C 0.000 }
gfCNCPoint5[10435] = {X 201.6473, Y 27.9611, Z -7.1667, A 0.000, B 0.000, C 0.000 }
gfCNCPoint5[10436] = {X 200.8675, Y 29.2352, Z -7.1667, A 0.000, B 0.000, C 0.000 }
gfCNCPoint5[10437] = {X 199.9328, Y 30.4003, Z -7.1667, A 0.000, B 0.000, C 0.000 }
gfCNCPoint5[10438] = {X 198.8581, Y 31.4376, Z -7.1667, A 0.000, B 0.000, C 0.000 }
gfCNCPoint5[10439] = {X 199.6409, Y 31.7994, Z -7.1667, A 0.000, B 0.000, C 0.000 }
gfCNCPoint5[10440] = {X 200.3381, Y 32.3070, Z -7.1667, A 0.000, B 0.000, C 0.000 }
gfCNCPoint5[10441] = {X 200.9230, Y 32.9407, Z -7.1667, A 0.000, B 0.000, C 0.000 }
gfCNCPoint5[10442] = {X 201.3730, Y 33.6764, Z -7.1667, A 0.000, B 0.000, C 0.000 }
gfCNCPoint5[10443] = {X 204.3942, Y 39.9182, Z -7.1667, A 0.000, B 0.000, C 0.000 }
gfCNCPoint5[10444] = {X 204.7207, Y 40.8441, Z -7.1667, A 0.000, B 0.000, C 0.000 }
gfCNCPoint5[10445] = {X 204.8337, Y 41.8194, Z -7.1667, A 0.000, B 0.000, C 0.000 }
gfCNCPoint5[10446] = {X 204.7276, Y 42.7955, Z -7.1667, A 0.000, B 0.000, C 0.000 }
gfCNCPoint5[10447] = {X 204.4078, Y 43.7238, Z -7.1667, A 0.000, B 0.000, C 0.000 }
gfCNCPoint5[10448] = {X 203.8900, Y 44.5580, Z -7.1667, A 0.000, B 0.000, C 0.000 }
gfCNCPoint5[10449] = {X 203.2002, Y 45.2567, Z -7.1667, A 0.000, B 0.000, C 0.000 }
gfCNCPoint5[10450] = {X 202.6640, Y 45.6902, Z -7.1667, A 0.000, B 0.000, C 0.000 }
gfCNCPoint5[10451] = {X 201.9527, Y 46.1594, Z -7.1667, A 0.000, B 0.000, C 0.000 }
gfCNCPoint5[10452] = {X 201.1645, Y 46.4832, Z -7.1667, A 0.000, B 0.000, C 0.000 }
gfCNCPoint5[10453] = {X 200.3287, Y 46.6495, Z -7.1667, A 0.000, B 0.000, C 0.000 }
gfCNCPoint5[10454] = {X 199.4765, Y 46.6520, Z -7.1667, A 0.000, B 0.000, C 0.000 }
gfCNCPoint5[10455] = {X 198.6398, Y 46.4907, Z -7.1667, A 0.000, B 0.000, C 0.000 }
gfCNCPoint5[10456] = {X 196.5325, Y 47.5871, Z -7.1667, A 0.000, B 0.000, C 0.000 }
gfCNCPoint5[10457] = {X 194.3411, Y 48.5043, Z -7.1667, A 0.000, B 0.000, C 0.000 }
gfCNCPoint5[10458] = {X 192.0811, Y 49.2359, Z -7.1667, A 0.000, B 0.000, C 0.000 }
gfCNCPoint5[10459] = {X 190.2778, Y 49.6715, Z -7.1667, A 0.000, B 0.000, C 0.000 }
gfCNCPoint5[10460] = {X 188.4447, Y 49.9570, Z -7.1667, A 0.000, B 0.000, C 0.000 }
gfCNCPoint5[10461] = {X 186.5943, Y 50.0904, Z -7.1667, A 0.000, B 0.000, C 0.000 }
gfCNCPoint5[10462] = {X 184.7393, Y 50.0709, Z -7.1667, A 0.000, B 0.000, C 0.000 }
gfCNCPoint5[10463] = {X 184.7144, Y 50.5503, Z -7.1667, A 0.000, B 0.000, C 0.000 }
gfCNCPoint5[10464] = {X 185.7098, Y 51.5036, Z -7.1667, A 0.000, B 0.000, C 0.000 }
gfCNCPoint5[10465] = {X 186.5597, Y 52.5886, Z -7.1667, A 0.000, B 0.000, C 0.000 }
gfCNCPoint5[10466] = {X 187.2468, Y 53.7833, Z -7.1667, A 0.000, B 0.000, C 0.000 }
gfCNCPoint5[10467] = {X 187.7798, Y 55.1350, Z -7.1667, A 0.000, B 0.000, C 0.000 }
gfCNCPoint5[10468] = {X 188.1045, Y 56.5512, Z -7.1667, A 0.000, B 0.000, C 0.000 }
gfCNCPoint5[10469] = {X 188.2135, Y 58.0000, Z -7.1667, A 0.000, B 0.000, C 0.000 }
gfCNCPoint5[10470] = {X 188.2132, Y 59.0140, Z -7.1667, A 0.000, B 0.000, C 0.000 }
gfCNCPoint5[10471] = {X 188.2027, Y 59.3923, Z -7.1667, A 0.000, B 0.000, C 0.000 }
gfCNCPoint5[10472] = {X 188.1774, Y 59.7698, Z -7.1667, A 0.000, B 0.000, C 0.000 }
gfCNCPoint5[10473] = {X 206.8501, Y 80.1539, Z -7.1667, A 0.000, B 0.000, C 0.000 }
gfCNCPoint5[10474] = {X 212.1592, Y 75.2905, Z -7.1667, A 0.000, B 0.000, C 0.000 }
gfCNCPoint5[10475] = {X 215.1958, Y 78.6053, Z -7.1667, A 0.000, B 0.000, C 0.000 }
gfCNCPoint5[10476] = {X 218.3257, Y 76.6003, Z -7.1667, A 0.000, B 0.000, C 0.000 }
gfCNCPoint5[10477] = {X 216.9987, Y 76.0796, Z -7.1667, A 0.000, B 0.000, C 0.000 }
gfCNCPoint5[10478] = {X 216.3738, Y 75.8857, Z -7.1667, A 0.000, B 0.000, C 0.000 }
gfCNCPoint5[10479] = {X 215.7249, Y 75.8032, Z -7.1667, A 0.000, B 0.000, C 0.000 }
gfCNCPoint5[10480] = {X 213.9283, Y 75.6422, Z -7.1667, A 0.000, B 0.000, C 0.000 }
gfCNCPoint5[10481] = {X 212.1592, Y 75.2905, Z -7.1667, A 0.000, B 0.000, C 0.000 }
gfCNCPoint5[10482] = {X 210.3895, Y 76.9116, Z -7.1667, A 0.000, B 0.000, C 0.000 }
gfCNCPoint5[10483] = {X 214.7901, Y 81.7155, Z -7.1667, A 0.000, B 0.000, C 0.000 }
gfCNCPoint5[10484] = {X 223.5805, Y 76.0842, Z -7.1667, A 0.000, B 0.000, C 0.000 }
gfCNCPoint5[10485] = {X 217.8873, Y 73.8501, Z -7.1667, A 0.000, B 0.000, C 0.000 }
gfCNCPoint5[10486] = {X 216.8702, Y 73.5376, Z -7.1667, A 0.000, B 0.000, C 0.000 }
gfCNCPoint5[10487] = {X 215.8145, Y 73.4049, Z -7.1667, A 0.000, B 0.000, C 0.000 }
gfCNCPoint5[10488] = {X 214.2716, Y 73.2669, Z -7.1667, A 0.000, B 0.000, C 0.000 }
gfCNCPoint5[10489] = {X 212.7523, Y 72.9649, Z -7.1667, A 0.000, B 0.000, C 0.000 }
gfCNCPoint5[10490] = {X 211.1539, Y 72.4570, Z -7.1667, A 0.000, B 0.000, C 0.000 }
gfCNCPoint5[10491] = {X 209.6249, Y 71.7677, Z -7.1667, A 0.000, B 0.000, C 0.000 }
gfCNCPoint5[10492] = {X 208.1859, Y 70.9061, Z -7.1667, A 0.000, B 0.000, C 0.000 }
gfCNCPoint5[10493] = {X 206.8561, Y 69.8840, Z -7.1667, A 0.000, B 0.000, C 0.000 }
gfCNCPoint5[10494] = {X 205.6535, Y 68.7149, Z -7.1667, A 0.000, B 0.000, C 0.000 }
gfCNCPoint5[10495] = {X 204.5941, Y 67.4146, Z -7.1667, A 0.000, B 0.000, C 0.000 }
gfCNCPoint5[10496] = {X 203.6922, Y 66.0006, Z -7.1667, A 0.000, B 0.000, C 0.000 }
gfCNCPoint5[10497] = {X 202.9598, Y 64.4917, Z -7.1667, A 0.000, B 0.000, C 0.000 }
gfCNCPoint5[10498] = {X 202.4069, Y 62.9083, Z -7.1667, A 0.000, B 0.000, C 0.000 }
gfCNCPoint5[10499] = {X 202.0407, Y 61.2715, Z -7.1667, A 0.000, B 0.000, C 0.000 }
gfCNCPoint5[10500] = {X 199.6722, Y 61.6590, Z -7.1667, A 0.000, B 0.000, C 0.000 }
gfCNCPoint5[10501] = {X 199.5095, Y 60.3406, Z -7.1667, A 0.000, B 0.000, C 0.000 }
gfCNCPoint5[10502] = {X 199.4510, Y 59.0136, Z -7.1667, A 0.000, B 0.000, C 0.000 }
gfCNCPoint5[10503] = {X 199.4508, Y 58.0000, Z -7.1667, A 0.000, B 0.000, C 0.000 }
gfCNCPoint5[10504] = {X 199.5411, Y 56.2568, Z -7.1667, A 0.000, B 0.000, C 0.000 }
gfCNCPoint5[10505] = {X 199.8108, Y 54.5322, Z -7.1667, A 0.000, B 0.000, C 0.000 }
gfCNCPoint5[10506] = {X 197.5975, Y 55.4822, Z -7.1667, A 0.000, B 0.000, C 0.000 }
gfCNCPoint5[10507] = {X 195.3259, Y 56.2828, Z -7.1667, A 0.000, B 0.000, C 0.000 }
gfCNCPoint5[10508] = {X 195.3577, Y 56.6291, Z -7.1667, A 0.000, B 0.000, C 0.000 }
gfCNCPoint5[10509] = {X 195.3824, Y 56.9760, Z -7.1667, A 0.000, B 0.000, C 0.000 }
gfCNCPoint5[10510] = {X 199.6722, Y 61.6590, Z -7.1667, A 0.000, B 0.000, C 0.000 }
gfCNCPoint5[10511] = {X 202.0407, Y 61.2715, Z -7.1667, A 0.000, B 0.000, C 0.000 }
gfCNCPoint5[10512] = {X 201.9014, Y 60.1432, Z -7.1667, A 0.000, B 0.000, C 0.000 }
gfCNCPoint5[10513] = {X 201.8510, Y 59.0073, Z -7.1667, A 0.000, B 0.000, C 0.000 }
gfCNCPoint5[10514] = {X 201.8508, Y 58.0000, Z -7.1667, A 0.000, B 0.000, C 0.000 }
gfCNCPoint5[10515] = {X 201.9282, Y 56.5047, Z -7.1667, A 0.000, B 0.000, C 0.000 }
gfCNCPoint5[10516] = {X 202.1597, Y 55.0253, Z -7.1667, A 0.000, B 0.000, C 0.000 }
gfCNCPoint5[10517] = {X 202.4964, Y 53.7246, Z -7.1667, A 0.000, B 0.000, C 0.000 }
gfCNCPoint5[10518] = {X 202.9522, Y 52.4607, Z -7.1667, A 0.000, B 0.000, C 0.000 }
gfCNCPoint5[10519] = {X 203.5232, Y 51.2445, Z -7.1667, A 0.000, B 0.000, C 0.000 }
gfCNCPoint5[10520] = {X 202.2642, Y 51.6560, Z -7.1667, A 0.000, B 0.000, C 0.000 }
gfCNCPoint5[10521] = {X 200.9609, Y 51.8920, Z -7.1667, A 0.000, B 0.000, C 0.000 }
gfCNCPoint5[10522] = {X 199.6375, Y 51.9481, Z -7.1667, A 0.000, B 0.000, C 0.000 }
gfCNCPoint5[10523] = {X 199.2159, Y 52.1567, Z -7.1667, A 0.000, B 0.000, C 0.000 }
gfCNCPoint5[10524] = {X 198.7914, Y 52.3595, Z -7.1667, A 0.000, B 0.000, C 0.000 }
gfCNCPoint5[10525] = {X 196.1935, Y 53.4488, Z -7.1667, A 0.000, B 0.000, C 0.000 }
gfCNCPoint5[10526] = {X 193.5138, Y 54.3178, Z -7.1667, A 0.000, B 0.000, C 0.000 }
gfCNCPoint5[10527] = {X 193.0576, Y 54.4436, Z -7.1667, A 0.000, B 0.000, C 0.000 }
gfCNCPoint5[10528] = {X 192.5993, Y 54.5616, Z -7.1667, A 0.000, B 0.000, C 0.000 }
gfCNCPoint5[10529] = {X 192.9061, Y 56.2401, Z -7.1667, A 0.000, B 0.000, C 0.000 }
gfCNCPoint5[10530] = {X 193.0134, Y 57.9429, Z -7.1667, A 0.000, B 0.000, C 0.000 }
gfCNCPoint5[10531] = {X 210.3895, Y 76.9116, Z -7.1667, A 0.000, B 0.000, C 0.000 }
gfCNCPoint5[10532] = {X 208.6198, Y 78.5328, Z -7.1667, A 0.000, B 0.000, C 0.000 }
gfCNCPoint5[10533] = {X 214.3843, Y 84.8256, Z -7.1667, A 0.000, B 0.000, C 0.000 }
gfCNCPoint5[10534] = {X 228.8353, Y 75.5680, Z -7.1667, A 0.000, B 0.000, C 0.000 }
gfCNCPoint5[10535] = {X 218.7739, Y 71.6198, Z -7.1667, A 0.000, B 0.000, C 0.000 }
gfCNCPoint5[10536] = {X 217.8426, Y 71.3056, Z -7.1667, A 0.000, B 0.000, C 0.000 }
gfCNCPoint5[10537] = {X 216.8815, Y 71.1003, Z -7.1667, A 0.000, B 0.000, C 0.000 }
gfCNCPoint5[10538] = {X 215.9031, Y 71.0065, Z -7.1667, A 0.000, B 0.000, C 0.000 }
gfCNCPoint5[10539] = {X 214.2336, Y 70.8306, Z -7.1667, A 0.000, B 0.000, C 0.000 }
gfCNCPoint5[10540] = {X 212.6046, Y 70.4250, Z -7.1667, A 0.000, B 0.000, C 0.000 }
gfCNCPoint5[10541] = {X 211.0476, Y 69.7975, Z -7.1667, A 0.000, B 0.000, C 0.000 }
gfCNCPoint5[10542] = {X 209.5926, Y 68.9602, Z -7.1667, A 0.000, B 0.000, C 0.000 }
gfCNCPoint5[10543] = {X 208.2677, Y 67.9292, Z -7.1667, A 0.000, B 0.000, C 0.000 }
gfCNCPoint5[10544] = {X 207.0985, Y 66.7245, Z -7.1667, A 0.000, B 0.000, C 0.000 }
gfCNCPoint5[10545] = {X 206.1077, Y 65.3694, Z -7.1667, A 0.000, B 0.000, C 0.000 }
gfCNCPoint5[10546] = {X 205.3142, Y 63.8900, Z -7.1667, A 0.000, B 0.000, C 0.000 }
gfCNCPoint5[10547] = {X 204.7335, Y 62.3149, Z -7.1667, A 0.000, B 0.000, C 0.000 }
gfCNCPoint5[10548] = {X 204.3768, Y 60.6745, Z -7.1667, A 0.000, B 0.000, C 0.000 }
gfCNCPoint5[10549] = {X 204.2510, Y 59.0005, Z -7.1667, A 0.000, B 0.000, C 0.000 }
gfCNCPoint5[10550] = {X 204.2508, Y 58.0000, Z -7.1667, A 0.000, B 0.000, C 0.000 }
gfCNCPoint5[10551] = {X 204.3396, Y 56.5378, Z -7.1667, A 0.000, B 0.000, C 0.000 }
gfCNCPoint5[10552] = {X 204.6048, Y 55.0970, Z -7.1667, A 0.000, B 0.000, C 0.000 }
gfCNCPoint5[10553] = {X 205.0424, Y 53.6990, Z -7.1667, A 0.000, B 0.000, C 0.000 }
gfCNCPoint5[10554] = {X 205.6460, Y 52.3642, Z -7.1667, A 0.000, B 0.000, C 0.000 }
gfCNCPoint5[10555] = {X 206.5296, Y 50.9387, Z -7.1667, A 0.000, B 0.000, C 0.000 }
gfCNCPoint5[10556] = {X 207.6020, Y 49.6493, Z -7.1667, A 0.000, B 0.000, C 0.000 }
gfCNCPoint5[10557] = {X 208.8427, Y 48.5209, Z -7.1667, A 0.000, B 0.000, C 0.000 }
gfCNCPoint5[10558] = {X 210.2277, Y 47.5751, Z -7.1667, A 0.000, B 0.000, C 0.000 }
gfCNCPoint5[10559] = {X 209.8801, Y 46.3328, Z -7.1667, A 0.000, B 0.000, C 0.000 }
gfCNCPoint5[10560] = {X 209.7572, Y 45.0487, Z -7.1667, A 0.000, B 0.000, C 0.000 }
gfCNCPoint5[10561] = {X 209.7570, Y 44.1909, Z -7.1667, A 0.000, B 0.000, C 0.000 }
gfCNCPoint5[10562] = {X 209.8558, Y 43.0023, Z -7.1667, A 0.000, B 0.000, C 0.000 }
gfCNCPoint5[10563] = {X 210.1494, Y 41.8463, Z -7.1667, A 0.000, B 0.000, C 0.000 }
gfCNCPoint5[10564] = {X 210.6298, Y 40.7546, Z -7.1667, A 0.000, B 0.000, C 0.000 }
gfCNCPoint5[10565] = {X 211.2839, Y 39.7572, Z -7.1667, A 0.000, B 0.000, C 0.000 }
gfCNCPoint5[10566] = {X 211.2839, Y 37.0748, Z -7.1667, A 0.000, B 0.000, C 0.000 }
gfCNCPoint5[10567] = {X 208.8839, Y 37.0748, Z -7.1667, A 0.000, B 0.000, C 0.000 }
gfCNCPoint5[10568] = {X 208.8839, Y 18.1961, Z -7.1667, A 0.000, B 0.000, C 0.000 }
gfCNCPoint5[10569] = {X 208.2323, Y 17.0004, Z -7.1667, A 0.000, B 0.000, C 0.000 }
gfCNCPoint5[10570] = {X 207.7550, Y 15.7251, Z -7.1667, A 0.000, B 0.000, C 0.000 }
gfCNCPoint5[10571] = {X 207.4614, Y 14.3955, Z -7.1667, A 0.000, B 0.000, C 0.000 }
gfCNCPoint5[10572] = {X 207.3572, Y 13.0378, Z -7.1667, A 0.000, B 0.000, C 0.000 }
gfCNCPoint5[10573] = {X 207.3570, Y 12.1868, Z -7.1667, A 0.000, B 0.000, C 0.000 }
gfCNCPoint5[10574] = {X 207.3580, Y 12.0458, Z -7.1667, A 0.000, B 0.000, C 0.000 }
gfCNCPoint5[10575] = {X 207.3611, Y 11.9049, Z -7.1667, A 0.000, B 0.000, C 0.000 }
gfCNCPoint5[10576] = {X 205.8582, Y 11.9049, Z -7.1667, A 0.000, B 0.000, C 0.000 }
gfCNCPoint5[10577] = {X 206.6133, Y 13.3418, Z -7.1667, A 0.000, B 0.000, C 0.000 }
gfCNCPoint5[10578] = {X 207.2387, Y 14.8398, Z -7.1667, A 0.000, B 0.000, C 0.000 }
gfCNCPoint5[10579] = {X 207.7994, Y 16.7126, Z -7.1667, A 0.000, B 0.000, C 0.000 }
gfCNCPoint5[10580] = {X 208.1782, Y 18.6305, Z -7.1667, A 0.000, B 0.000, C 0.000 }
gfCNCPoint5[10581] = {X 208.3716, Y 20.5759, Z -7.1667, A 0.000, B 0.000, C 0.000 }
gfCNCPoint5[10582] = {X 208.3776, Y 22.5309, Z -7.1667, A 0.000, B 0.000, C 0.000 }
gfCNCPoint5[10583] = {X 208.1964, Y 24.4774, Z -7.1667, A 0.000, B 0.000, C 0.000 }
gfCNCPoint5[10584] = {X 207.8295, Y 26.3977, Z -7.1667, A 0.000, B 0.000, C 0.000 }
gfCNCPoint5[10585] = {X 207.3622, Y 28.0103, Z -7.1667, A 0.000, B 0.000, C 0.000 }
gfCNCPoint5[10586] = {X 206.7387, Y 29.5692, Z -7.1667, A 0.000, B 0.000, C 0.000 }
gfCNCPoint5[10587] = {X 205.9649, Y 31.0592, Z -7.1667, A 0.000, B 0.000, C 0.000 }
gfCNCPoint5[10588] = {X 206.0467, Y 31.2169, Z -7.1667, A 0.000, B 0.000, C 0.000 }
gfCNCPoint5[10589] = {X 206.1255, Y 31.3760, Z -7.1667, A 0.000, B 0.000, C 0.000 }
gfCNCPoint5[10590] = {X 208.8839, Y 37.0748, Z -7.1667, A 0.000, B 0.000, C 0.000 }
gfCNCPoint5[10591] = {X 211.2839, Y 37.0748, Z -7.1667, A 0.000, B 0.000, C 0.000 }
gfCNCPoint5[10592] = {X 211.2836, Y 17.4386, Z -7.1667, A 0.000, B 0.000, C 0.000 }
gfCNCPoint5[10593] = {X 210.6356, Y 16.4450, Z -7.1667, A 0.000, B 0.000, C 0.000 }
gfCNCPoint5[10594] = {X 210.1575, Y 15.3595, Z -7.1667, A 0.000, B 0.000, C 0.000 }
gfCNCPoint5[10595] = {X 209.8621, Y 14.2106, Z -7.1667, A 0.000, B 0.000, C 0.000 }
gfCNCPoint5[10596] = {X 209.7572, Y 13.0291, Z -7.1667, A 0.000, B 0.000, C 0.000 }
gfCNCPoint5[10597] = {X 209.7570, Y 12.1868, Z -7.1667, A 0.000, B 0.000, C 0.000 }
gfCNCPoint5[10598] = {X 209.7578, Y 12.0808, Z -7.1667, A 0.000, B 0.000, C 0.000 }
gfCNCPoint5[10599] = {X 209.7601, Y 11.9748, Z -7.1667, A 0.000, B 0.000, C 0.000 }
gfCNCPoint5[10600] = {X 209.9068, Y 10.7176, Z -7.1667, A 0.000, B 0.000, C 0.000 }
gfCNCPoint5[10601] = {X 210.2690, Y 9.5049, Z -7.1667, A 0.000, B 0.000, C 0.000 }
gfCNCPoint5[10602] = {X 200.9088, Y 9.5049, Z -7.1667, A 0.000, B 0.000, C 0.000 }
gfCNCPoint5[10603] = {X 201.9824, Y 10.6133, Z -7.1667, A 0.000, B 0.000, C 0.000 }
gfCNCPoint5[10604] = {X 202.9441, Y 11.8201, Z -7.1667, A 0.000, B 0.000, C 0.000 }
gfCNCPoint5[10605] = {X 203.7850, Y 13.1140, Z -7.1667, A 0.000, B 0.000, C 0.000 }
gfCNCPoint5[10606] = {X 204.4384, Y 14.3567, Z -7.1667, A 0.000, B 0.000, C 0.000 }
gfCNCPoint5[10607] = {X 204.9802, Y 15.6519, Z -7.1667, A 0.000, B 0.000, C 0.000 }
gfCNCPoint5[10608] = {X 205.5526, Y 17.6384, Z -7.1667, A 0.000, B 0.000, C 0.000 }
gfCNCPoint5[10609] = {X 205.8933, Y 19.6775, Z -7.1667, A 0.000, B 0.000, C 0.000 }
gfCNCPoint5[10610] = {X 205.9977, Y 21.7422, Z -7.1667, A 0.000, B 0.000, C 0.000 }
gfCNCPoint5[10611] = {X 205.8644, Y 23.8053, Z -7.1667, A 0.000, B 0.000, C 0.000 }
gfCNCPoint5[10612] = {X 205.4953, Y 25.8394, Z -7.1667, A 0.000, B 0.000, C 0.000 }
gfCNCPoint5[10613] = {X 205.0941, Y 27.2258, Z -7.1667, A 0.000, B 0.000, C 0.000 }
gfCNCPoint5[10614] = {X 204.5584, Y 28.5660, Z -7.1667, A 0.000, B 0.000, C 0.000 }
gfCNCPoint5[10615] = {X 203.8936, Y 29.8471, Z -7.1667, A 0.000, B 0.000, C 0.000 }
gfCNCPoint5[10616] = {X 203.1059, Y 31.0565, Z -7.1667, A 0.000, B 0.000, C 0.000 }
gfCNCPoint5[10617] = {X 203.5735, Y 31.7152, Z -7.1667, A 0.000, B 0.000, C 0.000 }
gfCNCPoint5[10618] = {X 203.9653, Y 32.4217, Z -7.1667, A 0.000, B 0.000, C 0.000 }
gfCNCPoint5[10619] = {X 206.9865, Y 38.6634, Z -7.1667, A 0.000, B 0.000, C 0.000 }
gfCNCPoint5[10620] = {X 207.4240, Y 39.8017, Z -7.1667, A 0.000, B 0.000, C 0.000 }
gfCNCPoint5[10621] = {X 207.6653, Y 40.9971, Z -7.1667, A 0.000, B 0.000, C 0.000 }
gfCNCPoint5[10622] = {X 207.7038, Y 42.2159, Z -7.1667, A 0.000, B 0.000, C 0.000 }
gfCNCPoint5[10623] = {X 207.5382, Y 43.4241, Z -7.1667, A 0.000, B 0.000, C 0.000 }
gfCNCPoint5[10624] = {X 207.1733, Y 44.5877, Z -7.1667, A 0.000, B 0.000, C 0.000 }
gfCNCPoint5[10625] = {X 206.6193, Y 45.6741, Z -7.1667, A 0.000, B 0.000, C 0.000 }
gfCNCPoint5[10626] = {X 205.8917, Y 46.6527, Z -7.1667, A 0.000, B 0.000, C 0.000 }
gfCNCPoint5[10627] = {X 205.0110, Y 47.4962, Z -7.1667, A 0.000, B 0.000, C 0.000 }
gfCNCPoint5[10628] = {X 204.4746, Y 47.9298, Z -7.1667, A 0.000, B 0.000, C 0.000 }
gfCNCPoint5[10629] = {X 203.5894, Y 48.5432, Z -7.1667, A 0.000, B 0.000, C 0.000 }
gfCNCPoint5[10630] = {X 202.6236, Y 49.0195, Z -7.1667, A 0.000, B 0.000, C 0.000 }
gfCNCPoint5[10631] = {X 201.4897, Y 49.3737, Z -7.1667, A 0.000, B 0.000, C 0.000 }
gfCNCPoint5[10632] = {X 200.3134, Y 49.5390, Z -7.1667, A 0.000, B 0.000, C 0.000 }
gfCNCPoint5[10633] = {X 199.1259, Y 49.5112, Z -7.1667, A 0.000, B 0.000, C 0.000 }
gfCNCPoint5[10634] = {X 197.0997, Y 50.4926, Z -7.1667, A 0.000, B 0.000, C 0.000 }
gfCNCPoint5[10635] = {X 195.0083, Y 51.3263, Z -7.1667, A 0.000, B 0.000, C 0.000 }
gfCNCPoint5[10636] = {X 192.8626, Y 52.0078, Z -7.1667, A 0.000, B 0.000, C 0.000 }
gfCNCPoint5[10637] = {X 192.4426, Y 52.1237, Z -7.1667, A 0.000, B 0.000, C 0.000 }
gfCNCPoint5[10638] = {X 192.0206, Y 52.2324, Z -7.1667, A 0.000, B 0.000, C 0.000 }
gfCNCPoint5[10639] = {X 190.7205, Y 52.5195, Z -7.1667, A 0.000, B 0.000, C 0.000 }
gfCNCPoint5[10640] = {X 189.4072, Y 52.7379, Z -7.1667, A 0.000, B 0.000, C 0.000 }
gfCNCPoint5[10641] = {X 189.9008, Y 53.9120, Z -7.1667, A 0.000, B 0.000, C 0.000 }
gfCNCPoint5[10642] = {X 190.2680, Y 55.1315, Z -7.1667, A 0.000, B 0.000, C 0.000 }
gfCNCPoint5[10643] = {X 190.5268, Y 56.5554, Z -7.1667, A 0.000, B 0.000, C 0.000 }
gfCNCPoint5[10644] = {X 190.6135, Y 58.0000, Z -7.1667, A 0.000, B 0.000, C 0.000 }
gfCNCPoint5[10645] = {X 190.6132, Y 58.8758, Z -7.1667, A 0.000, B 0.000, C 0.000 }
gfCNCPoint5[10646] = {X 208.6198, Y 78.5328, Z -7.1667, A 0.000, B 0.000, C 0.000 }
gfCNCPoint5[10647] = {X 206.8501, Y 80.1539, Z -7.1667, A 0.000, B 0.000, C 0.000 }
gfCNCPoint5[10648] = {X 213.2488, Y 87.1391, Z -7.1667, A 0.000, B 0.000, C 0.000 }
gfCNCPoint5[10649] = {X 213.3847, Y 87.2852, Z -7.1667, A 0.000, B 0.000, C 0.000 }
gfCNCPoint5[10650] = {X 213.5229, Y 87.4293, Z -7.1667, A 0.000, B 0.000, C 0.000 }
gfCNCPoint5[10651] = {X 214.2173, Y 87.3791, Z -7.1667, A 0.000, B 0.000, C 0.000 }
gfCNCPoint5[10652] = {X 214.9122, Y 87.3377, Z -7.1667, A 0.000, B 0.000, C 0.000 }
gfCNCPoint5[10653] = {X 234.0902, Y 75.0519, Z -7.1667, A 0.000, B 0.000, C 0.000 }
gfCNCPoint5[10654] = {X 219.6594, Y 69.3891, Z -7.1667, A 0.000, B 0.000, C 0.000 }
gfCNCPoint5[10655] = {X 218.4692, Y 68.9888, Z -7.1667, A 0.000, B 0.000, C 0.000 }
gfCNCPoint5[10656] = {X 217.2410, Y 68.7273, Z -7.1667, A 0.000, B 0.000, C 0.000 }
gfCNCPoint5[10657] = {X 215.9909, Y 68.6081, Z -7.1667, A 0.000, B 0.000, C 0.000 }
gfCNCPoint5[10658] = {X 214.5209, Y 68.4434, Z -7.1667, A 0.000, B 0.000, C 0.000 }
gfCNCPoint5[10659] = {X 213.0932, Y 68.0566, Z -7.1667, A 0.000, B 0.000, C 0.000 }
gfCNCPoint5[10660] = {X 211.7411, Y 67.4568, Z -7.1667, A 0.000, B 0.000, C 0.000 }
gfCNCPoint5[10661] = {X 210.4961, Y 66.6580, Z -7.1667, A 0.000, B 0.000, C 0.000 }
gfCNCPoint5[10662] = {X 209.3874, Y 65.6788, Z -7.1667, A 0.000, B 0.000, C 0.000 }
gfCNCPoint5[10663] = {X 208.4408, Y 64.5421, Z -7.1667, A 0.000, B 0.000, C 0.000 }
gfCNCPoint5[10664] = {X 207.6785, Y 63.2745, Z -7.1667, A 0.000, B 0.000, C 0.000 }
gfCNCPoint5[10665] = {X 207.1182, Y 61.9055, Z -7.1667, A 0.000, B 0.000, C 0.000 }
gfCNCPoint5[10666] = {X 206.7730, Y 60.4672, Z -7.1667, A 0.000, B 0.000, C 0.000 }
gfCNCPoint5[10667] = {X 206.6510, Y 58.9930, Z -7.1667, A 0.000, B 0.000, C 0.000 }
gfCNCPoint5[10668] = {X 206.6508, Y 58.0000, Z -7.1667, A 0.000, B 0.000, C 0.000 }
gfCNCPoint5[10669] = {X 206.7577, Y 56.5655, Z -7.1667, A 0.000, B 0.000, C 0.000 }
gfCNCPoint5[10670] = {X 207.0759, Y 55.1628, Z -7.1667, A 0.000, B 0.000, C 0.000 }
gfCNCPoint5[10671] = {X 207.5986, Y 53.8226, Z -7.1667, A 0.000, B 0.000, C 0.000 }
gfCNCPoint5[10672] = {X 208.3140, Y 52.5747, Z -7.1667, A 0.000, B 0.000, C 0.000 }
gfCNCPoint5[10673] = {X 209.2065, Y 51.4466, Z -7.1667, A 0.000, B 0.000, C 0.000 }
gfCNCPoint5[10674] = {X 210.2563, Y 50.4632, Z -7.1667, A 0.000, B 0.000, C 0.000 }
gfCNCPoint5[10675] = {X 211.4402, Y 49.6463, Z -7.1667, A 0.000, B 0.000, C 0.000 }
gfCNCPoint5[10676] = {X 212.5893, Y 49.0723, Z -7.1667, A 0.000, B 0.000, C 0.000 }
gfCNCPoint5[10677] = {X 213.8042, Y 48.6556, Z -7.1667, A 0.000, B 0.000, C 0.000 }
gfCNCPoint5[10678] = {X 213.2578, Y 48.0874, Z -7.1667, A 0.000, B 0.000, C 0.000 }
gfCNCPoint5[10679] = {X 212.8100, Y 47.4386, Z -7.1667, A 0.000, B 0.000, C 0.000 }
gfCNCPoint5[10680] = {X 212.4725, Y 46.7262, Z -7.1667, A 0.000, B 0.000, C 0.000 }
gfCNCPoint5[10681] = {X 212.2401, Y 45.8965, Z -7.1667, A 0.000, B 0.000, C 0.000 }
gfCNCPoint5[10682] = {X 212.1572, Y 45.0389, Z -7.1667, A 0.000, B 0.000, C 0.000 }
gfCNCPoint5[10683] = {X 212.1570, Y 44.1909, Z -7.1667, A 0.000, B 0.000, C 0.000 }
gfCNCPoint5[10684] = {X 212.2382, Y 43.3120, Z -7.1667, A 0.000, B 0.000, C 0.000 }
gfCNCPoint5[10685] = {X 212.4788, Y 42.4628, Z -7.1667, A 0.000, B 0.000, C 0.000 }
gfCNCPoint5[10686] = {X 212.8709, Y 41.6720, Z -7.1667, A 0.000, B 0.000, C 0.000 }
gfCNCPoint5[10687] = {X 213.4011, Y 40.9664, Z -7.1667, A 0.000, B 0.000, C 0.000 }
gfCNCPoint5[10688] = {X 213.6811, Y 40.6575, Z -7.1667, A 0.000, B 0.000, C 0.000 }
gfCNCPoint5[10689] = {X 213.6839, Y 40.3041, Z -7.1667, A 0.000, B 0.000, C 0.000 }
gfCNCPoint5[10690] = {X 213.6839, Y 17.4645, Z -7.1667, A 0.000, B 0.000, C 0.000 }
gfCNCPoint5[10691] = {X 213.6785, Y 16.7695, Z -7.1667, A 0.000, B 0.000, C 0.000 }
gfCNCPoint5[10692] = {X 213.6783, Y 16.5183, Z -7.1667, A 0.000, B 0.000, C 0.000 }
gfCNCPoint5[10693] = {X 213.0396, Y 15.7771, Z -7.1667, A 0.000, B 0.000, C 0.000 }
gfCNCPoint5[10694] = {X 212.5615, Y 14.9234, Z -7.1667, A 0.000, B 0.000, C 0.000 }
gfCNCPoint5[10695] = {X 212.2634, Y 13.9915, Z -7.1667, A 0.000, B 0.000, C 0.000 }
gfCNCPoint5[10696] = {X 212.1572, Y 13.0188, Z -7.1667, A 0.000, B 0.000, C 0.000 }
gfCNCPoint5[10697] = {X 212.1570, Y 12.1868, Z -7.1667, A 0.000, B 0.000, C 0.000 }
gfCNCPoint5[10698] = {X 212.2436, Y 11.2717, Z -7.1667, A 0.000, B 0.000, C 0.000 }
gfCNCPoint5[10699] = {X 212.5002, Y 10.3890, Z -7.1667, A 0.000, B 0.000, C 0.000 }
gfCNCPoint5[10700] = {X 212.9450, Y 9.5280, Z -7.1667, A 0.000, B 0.000, C 0.000 }
gfCNCPoint5[10701] = {X 213.5511, Y 8.7718, Z -7.1667, A 0.000, B 0.000, C 0.000 }
gfCNCPoint5[10702] = {X 214.2946, Y 8.1503, Z -7.1667, A 0.000, B 0.000, C 0.000 }
gfCNCPoint5[10703] = {X 215.1464, Y 7.6879, Z -7.1667, A 0.000, B 0.000, C 0.000 }
gfCNCPoint5[10704] = {X 216.0727, Y 7.4030, Z -7.1667, A 0.000, B 0.000, C 0.000 }
gfCNCPoint5[10705] = {X 217.0370, Y 7.3068, Z -7.1667, A 0.000, B 0.000, C 0.000 }
gfCNCPoint5[10706] = {X 223.4805, Y 7.3068, Z -7.1667, A 0.000, B 0.000, C 0.000 }
gfCNCPoint5[10707] = {X 224.4448, Y 7.4030, Z -7.1667, A 0.000, B 0.000, C 0.000 }
gfCNCPoint5[10708] = {X 225.3711, Y 7.6879, Z -7.1667, A 0.000, B 0.000, C 0.000 }
gfCNCPoint5[10709] = {X 226.2229, Y 8.1503, Z -7.1667, A 0.000, B 0.000, C 0.000 }
gfCNCPoint5[10710] = {X 226.9664, Y 8.7718, Z -7.1667, A 0.000, B 0.000, C 0.000 }
gfCNCPoint5[10711] = {X 227.5725, Y 9.5280, Z -7.1667, A 0.000, B 0.000, C 0.000 }
gfCNCPoint5[10712] = {X 228.0173, Y 10.3890, Z -7.1667, A 0.000, B 0.000, C 0.000 }
gfCNCPoint5[10713] = {X 228.2739, Y 11.2717, Z -7.1667, A 0.000, B 0.000, C 0.000 }
gfCNCPoint5[10714] = {X 228.3605, Y 12.1868, Z -7.1667, A 0.000, B 0.000, C 0.000 }
gfCNCPoint5[10715] = {X 228.3603, Y 13.0237, Z -7.1667, A 0.000, B 0.000, C 0.000 }
gfCNCPoint5[10716] = {X 228.2530, Y 13.9968, Z -7.1667, A 0.000, B 0.000, C 0.000 }
gfCNCPoint5[10717] = {X 227.9536, Y 14.9288, Z -7.1667, A 0.000, B 0.000, C 0.000 }
gfCNCPoint5[10718] = {X 227.4742, Y 15.7824, Z -7.1667, A 0.000, B 0.000, C 0.000 }
gfCNCPoint5[10719] = {X 226.8342, Y 16.5231, Z -7.1667, A 0.000, B 0.000, C 0.000 }
gfCNCPoint5[10720] = {X 226.8345, Y 25.8601, Z -7.1667, A 0.000, B 0.000, C 0.000 }
gfCNCPoint5[10721] = {X 231.6345, Y 25.8599, Z -7.1667, A 0.000, B 0.000, C 0.000 }
gfCNCPoint5[10722] = {X 231.6350, Y 38.9928, Z -7.1667, A 0.000, B 0.000, C 0.000 }
gfCNCPoint5[10723] = {X 231.6440, Y 39.0069, Z -7.1667, A 0.000, B 0.000, C 0.000 }
gfCNCPoint5[10724] = {X 232.3931, Y 37.9855, Z -7.1667, A 0.000, B 0.000, C 0.000 }
gfCNCPoint5[10725] = {X 233.2692, Y 37.0706, Z -7.1667, A 0.000, B 0.000, C 0.000 }
gfCNCPoint5[10726] = {X 234.2573, Y 36.2780, Z -7.1667, A 0.000, B 0.000, C 0.000 }
gfCNCPoint5[10727] = {X 235.5690, Y 33.7105, Z -7.1667, A 0.000, B 0.000, C 0.000 }
gfCNCPoint5[10728] = {X 234.4281, Y 32.2862, Z -7.1667, A 0.000, B 0.000, C 0.000 }
gfCNCPoint5[10729] = {X 233.4496, Y 30.7458, Z -7.1667, A 0.000, B 0.000, C 0.000 }
gfCNCPoint5[10730] = {X 232.6453, Y 29.1077, Z -7.1667, A 0.000, B 0.000, C 0.000 }
gfCNCPoint5[10731] = {X 232.0246, Y 27.3916, Z -7.1667, A 0.000, B 0.000, C 0.000 }
gfCNCPoint5[10732] = {X 231.8157, Y 26.6293, Z -7.1667, A 0.000, B 0.000, C 0.000 }
gfCNCPoint5[10733] = {X 231.6345, Y 25.8599, Z -7.1667, A 0.000, B 0.000, C 0.000 }
gfCNCPoint5[10734] = {X 229.2345, Y 25.8600, Z -7.1667, A 0.000, B 0.000, C 0.000 }
gfCNCPoint5[10735] = {X 229.2350, Y 39.7497, Z -7.1667, A 0.000, B 0.000, C 0.000 }
gfCNCPoint5[10736] = {X 229.4338, Y 40.0187, Z -7.1667, A 0.000, B 0.000, C 0.000 }
gfCNCPoint5[10737] = {X 229.6200, Y 40.2966, Z -7.1667, A 0.000, B 0.000, C 0.000 }
gfCNCPoint5[10738] = {X 230.1055, Y 41.1910, Z -7.1667, A 0.000, B 0.000, C 0.000 }
gfCNCPoint5[10739] = {X 230.4616, Y 42.1443, Z -7.1667, A 0.000, B 0.000, C 0.000 }
gfCNCPoint5[10740] = {X 230.6813, Y 43.1379, Z -7.1667, A 0.000, B 0.000, C 0.000 }
gfCNCPoint5[10741] = {X 230.7603, Y 44.1524, Z -7.1667, A 0.000, B 0.000, C 0.000 }
gfCNCPoint5[10742] = {X 230.7605, Y 45.0000, Z -7.1667, A 0.000, B 0.000, C 0.000 }
gfCNCPoint5[10743] = {X 230.7459, Y 45.4609, Z -7.1667, A 0.000, B 0.000, C 0.000 }
gfCNCPoint5[10744] = {X 230.7021, Y 45.9200, Z -7.1667, A 0.000, B 0.000, C 0.000 }
gfCNCPoint5[10745] = {X 232.5859, Y 45.9200, Z -7.1667, A 0.000, B 0.000, C 0.000 }
gfCNCPoint5[10746] = {X 232.5421, Y 45.4609, Z -7.1667, A 0.000, B 0.000, C 0.000 }
gfCNCPoint5[10747] = {X 232.5275, Y 45.0000, Z -7.1667, A 0.000, B 0.000, C 0.000 }
gfCNCPoint5[10748] = {X 232.5275, Y 44.2089, Z -7.1667, A 0.000, B 0.000, C 0.000 }
gfCNCPoint5[10749] = {X 232.6006, Y 43.1798, Z -7.1667, A 0.000, B 0.000, C 0.000 }
gfCNCPoint5[10750] = {X 232.8184, Y 42.1713, Z -7.1667, A 0.000, B 0.000, C 0.000 }
gfCNCPoint5[10751] = {X 233.1766, Y 41.2038, Z -7.1667, A 0.000, B 0.000, C 0.000 }
gfCNCPoint5[10752] = {X 233.6680, Y 40.2966, Z -7.1667, A 0.000, B 0.000, C 0.000 }
gfCNCPoint5[10753] = {X 234.3527, Y 39.3876, Z -7.1667, A 0.000, B 0.000, C 0.000 }
gfCNCPoint5[10754] = {X 235.1707, Y 38.5964, Z -7.1667, A 0.000, B 0.000, C 0.000 }
gfCNCPoint5[10755] = {X 236.1021, Y 37.9424, Z -7.1667, A 0.000, B 0.000, C 0.000 }
gfCNCPoint5[10756] = {X 238.4996, Y 33.2494, Z -7.1667, A 0.000, B 0.000, C 0.000 }
gfCNCPoint5[10757] = {X 237.3858, Y 32.1416, Z -7.1667, A 0.000, B 0.000, C 0.000 }
gfCNCPoint5[10758] = {X 236.4003, Y 30.9181, Z -7.1667, A 0.000, B 0.000, C 0.000 }
gfCNCPoint5[10759] = {X 235.5552, Y 29.5937, Z -7.1667, A 0.000, B 0.000, C 0.000 }
gfCNCPoint5[10760] = {X 234.8607, Y 28.1846, Z -7.1667, A 0.000, B 0.000, C 0.000 }
gfCNCPoint5[10761] = {X 234.3251, Y 26.7077, Z -7.1667, A 0.000, B 0.000, C 0.000 }
gfCNCPoint5[10762] = {X 234.1405, Y 26.0329, Z -7.1667, A 0.000, B 0.000, C 0.000 }
gfCNCPoint5[10763] = {X 233.9801, Y 25.3519, Z -7.1667, A 0.000, B 0.000, C 0.000 }
gfCNCPoint5[10764] = {X 233.6671, Y 23.4618, Z -7.1667, A 0.000, B 0.000, C 0.000 }
gfCNCPoint5[10765] = {X 233.5411, Y 21.5501, Z -7.1667, A 0.000, B 0.000, C 0.000 }
gfCNCPoint5[10766] = {X 233.6034, Y 19.6353, Z -7.1667, A 0.000, B 0.000, C 0.000 }
gfCNCPoint5[10767] = {X 233.8533, Y 17.7358, Z -7.1667, A 0.000, B 0.000, C 0.000 }
gfCNCPoint5[10768] = {X 234.2884, Y 15.8700, Z -7.1667, A 0.000, B 0.000, C 0.000 }
gfCNCPoint5[10769] = {X 234.7347, Y 14.5417, Z -7.1667, A 0.000, B 0.000, C 0.000 }
gfCNCPoint5[10770] = {X 235.3045, Y 13.2614, Z -7.1667, A 0.000, B 0.000, C 0.000 }
gfCNCPoint5[10771] = {X 233.1605, Y 12.1829, Z -7.1667, A 0.000, B 0.000, C 0.000 }
gfCNCPoint5[10772] = {X 233.2314, Y 12.0436, Z -7.1667, A 0.000, B 0.000, C 0.000 }
gfCNCPoint5[10773] = {X 233.3035, Y 11.9049, Z -7.1667, A 0.000, B 0.000, C 0.000 }
gfCNCPoint5[10774] = {X 233.1564, Y 11.9049, Z -7.1667, A 0.000, B 0.000, C 0.000 }
gfCNCPoint5[10775] = {X 233.1594, Y 12.0439, Z -7.1667, A 0.000, B 0.000, C 0.000 }
gfCNCPoint5[10776] = {X 233.1605, Y 12.1829, Z -7.1667, A 0.000, B 0.000, C 0.000 }
gfCNCPoint5[10777] = {X 235.3045, Y 13.2614, Z -7.1667, A 0.000, B 0.000, C 0.000 }
gfCNCPoint5[10778] = {X 235.3655, Y 13.1415, Z -7.1667, A 0.000, B 0.000, C 0.000 }
gfCNCPoint5[10779] = {X 235.4276, Y 13.0222, Z -7.1667, A 0.000, B 0.000, C 0.000 }
gfCNCPoint5[10780] = {X 236.1689, Y 11.7670, Z -7.1667, A 0.000, B 0.000, C 0.000 }
gfCNCPoint5[10781] = {X 237.0300, Y 10.5907, Z -7.1667, A 0.000, B 0.000, C 0.000 }
gfCNCPoint5[10782] = {X 238.0026, Y 9.5049, Z -7.1667, A 0.000, B 0.000, C 0.000 }
gfCNCPoint5[10783] = {X 230.2485, Y 9.5049, Z -7.1667, A 0.000, B 0.000, C 0.000 }
gfCNCPoint5[10784] = {X 230.6107, Y 10.7176, Z -7.1667, A 0.000, B 0.000, C 0.000 }
gfCNCPoint5[10785] = {X 230.7574, Y 11.9748, Z -7.1667, A 0.000, B 0.000, C 0.000 }
gfCNCPoint5[10786] = {X 230.7597, Y 12.0808, Z -7.1667, A 0.000, B 0.000, C 0.000 }
gfCNCPoint5[10787] = {X 230.7605, Y 12.1868, Z -7.1667, A 0.000, B 0.000, C 0.000 }
gfCNCPoint5[10788] = {X 230.7602, Y 13.0462, Z -7.1667, A 0.000, B 0.000, C 0.000 }
gfCNCPoint5[10789] = {X 230.6532, Y 14.2231, Z -7.1667, A 0.000, B 0.000, C 0.000 }
gfCNCPoint5[10790] = {X 230.3572, Y 15.3673, Z -7.1667, A 0.000, B 0.000, C 0.000 }
gfCNCPoint5[10791] = {X 229.8800, Y 16.4485, Z -7.1667, A 0.000, B 0.000, C 0.000 }
gfCNCPoint5[10792] = {X 229.2342, Y 17.4382, Z -7.1667, A 0.000, B 0.000, C 0.000 }
gfCNCPoint5[10793] = {X 229.2345, Y 25.8600, Z -7.1667, A 0.000, B 0.000, C 0.000 }
gfCNCPoint5[10794] = {X 226.8345, Y 25.8601, Z -7.1667, A 0.000, B 0.000, C 0.000 }
gfCNCPoint5[10795] = {X 226.8351, Y 40.6646, Z -7.1667, A 0.000, B 0.000, C 0.000 }
gfCNCPoint5[10796] = {X 227.4749, Y 41.4054, Z -7.1667, A 0.000, B 0.000, C 0.000 }
gfCNCPoint5[10797] = {X 227.9540, Y 42.2589, Z -7.1667, A 0.000, B 0.000, C 0.000 }
gfCNCPoint5[10798] = {X 228.2531, Y 43.1909, Z -7.1667, A 0.000, B 0.000, C 0.000 }
gfCNCPoint5[10799] = {X 228.3603, Y 44.1638, Z -7.1667, A 0.000, B 0.000, C 0.000 }
gfCNCPoint5[10800] = {X 228.3605, Y 45.0000, Z -7.1667, A 0.000, B 0.000, C 0.000 }
gfCNCPoint5[10801] = {X 228.3507, Y 45.3090, Z -7.1667, A 0.000, B 0.000, C 0.000 }
gfCNCPoint5[10802] = {X 228.3214, Y 45.6167, Z -7.1667, A 0.000, B 0.000, C 0.000 }
gfCNCPoint5[10803] = {X 228.0910, Y 46.5992, Z -7.1667, A 0.000, B 0.000, C 0.000 }
gfCNCPoint5[10804] = {X 227.6635, Y 47.5134, Z -7.1667, A 0.000, B 0.000, C 0.000 }
gfCNCPoint5[10805] = {X 227.0571, Y 48.3200, Z -7.1667, A 0.000, B 0.000, C 0.000 }
gfCNCPoint5[10806] = {X 226.7053, Y 47.9934, Z -7.1667, A 0.000, B 0.000, C 0.000 }
gfCNCPoint5[10807] = {X 226.0261, Y 48.5889, Z -7.1667, A 0.000, B 0.000, C 0.000 }
gfCNCPoint5[10808] = {X 225.2396, Y 49.0331, Z -7.1667, A 0.000, B 0.000, C 0.000 }
gfCNCPoint5[10809] = {X 224.3790, Y 49.3073, Z -7.1667, A 0.000, B 0.000, C 0.000 }
gfCNCPoint5[10810] = {X 223.4805, Y 49.4000, Z -7.1667, A 0.000, B 0.000, C 0.000 }
gfCNCPoint5[10811] = {X 217.0370, Y 49.4000, Z -7.1667, A 0.000, B 0.000, C 0.000 }
gfCNCPoint5[10812] = {X 216.0579, Y 49.2897, Z -7.1667, A 0.000, B 0.000, C 0.000 }
gfCNCPoint5[10813] = {X 215.1279, Y 48.9643, Z -7.1667, A 0.000, B 0.000, C 0.000 }
gfCNCPoint5[10814] = {X 214.2937, Y 48.4401, Z -7.1667, A 0.000, B 0.000, C 0.000 }
gfCNCPoint5[10815] = {X 213.5969, Y 47.7433, Z -7.1667, A 0.000, B 0.000, C 0.000 }
gfCNCPoint5[10816] = {X 213.0727, Y 46.9091, Z -7.1667, A 0.000, B 0.000, C 0.000 }
gfCNCPoint5[10817] = {X 212.7473, Y 45.9791, Z -7.1667, A 0.000, B 0.000, C 0.000 }
gfCNCPoint5[10818] = {X 212.6370, Y 45.0000, Z -7.1667, A 0.000, B 0.000, C 0.000 }
gfCNCPoint5[10819] = {X 212.6370, Y 44.1909, Z -7.1667, A 0.000, B 0.000, C 0.000 }
gfCNCPoint5[10820] = {X 212.7100, Y 43.3999, Z -7.1667, A 0.000, B 0.000, C 0.000 }
gfCNCPoint5[10821] = {X 212.9266, Y 42.6356, Z -7.1667, A 0.000, B 0.000, C 0.000 }
gfCNCPoint5[10822] = {X 213.2795, Y 41.9239, Z -7.1667, A 0.000, B 0.000, C 0.000 }
gfCNCPoint5[10823] = {X 213.7567, Y 41.2888, Z -7.1667, A 0.000, B 0.000, C 0.000 }
gfCNCPoint5[10824] = {X 214.1597, Y 40.8442, Z -7.1667, A 0.000, B 0.000, C 0.000 }
gfCNCPoint5[10825] = {X 214.1639, Y 40.3060, Z -7.1667, A 0.000, B 0.000, C 0.000 }
gfCNCPoint5[10826] = {X 214.1639, Y 17.4626, Z -7.1667, A 0.000, B 0.000, C 0.000 }
gfCNCPoint5[10827] = {X 214.1585, Y 16.7691, Z -7.1667, A 0.000, B 0.000, C 0.000 }
gfCNCPoint5[10828] = {X 214.1581, Y 16.3055, Z -7.1667, A 0.000, B 0.000, C 0.000 }
gfCNCPoint5[10829] = {X 213.5161, Y 15.6168, Z -7.1667, A 0.000, B 0.000, C 0.000 }
gfCNCPoint5[10830] = {X 213.0353, Y 14.8073, Z -7.1667, A 0.000, B 0.000, C 0.000 }
gfCNCPoint5[10831] = {X 212.7377, Y 13.9141, Z -7.1667, A 0.000, B 0.000, C 0.000 }
gfCNCPoint5[10832] = {X 212.6370, Y 12.9780, Z -7.1667, A 0.000, B 0.000, C 0.000 }
gfCNCPoint5[10833] = {X 212.6370, Y 12.1868, Z -7.1667, A 0.000, B 0.000, C 0.000 }
gfCNCPoint5[10834] = {X 212.7473, Y 11.2077, Z -7.1667, A 0.000, B 0.000, C 0.000 }
gfCNCPoint5[10835] = {X 213.0728, Y 10.2777, Z -7.1667, A 0.000, B 0.000, C 0.000 }
gfCNCPoint5[10836] = {X 213.5970, Y 9.4435, Z -7.1667, A 0.000, B 0.000, C 0.000 }
gfCNCPoint5[10837] = {X 214.2937, Y 8.7468, Z -7.1667, A 0.000, B 0.000, C 0.000 }
gfCNCPoint5[10838] = {X 215.1279, Y 8.2226, Z -7.1667, A 0.000, B 0.000, C 0.000 }
gfCNCPoint5[10839] = {X 216.0579, Y 7.8971, Z -7.1667, A 0.000, B 0.000, C 0.000 }
gfCNCPoint5[10840] = {X 217.0370, Y 7.7868, Z -7.1667, A 0.000, B 0.000, C 0.000 }
gfCNCPoint5[10841] = {X 223.4805, Y 7.7868, Z -7.1667, A 0.000, B 0.000, C 0.000 }
gfCNCPoint5[10842] = {X 224.4596, Y 7.8971, Z -7.1667, A 0.000, B 0.000, C 0.000 }
gfCNCPoint5[10843] = {X 225.3896, Y 8.2226, Z -7.1667, A 0.000, B 0.000, C 0.000 }
gfCNCPoint5[10844] = {X 226.2238, Y 8.7468, Z -7.1667, A 0.000, B 0.000, C 0.000 }
gfCNCPoint5[10845] = {X 226.9205, Y 9.4435, Z -7.1667, A 0.000, B 0.000, C 0.000 }
gfCNCPoint5[10846] = {X 227.4447, Y 10.2777, Z -7.1667, A 0.000, B 0.000, C 0.000 }
gfCNCPoint5[10847] = {X 227.7702, Y 11.2077, Z -7.1667, A 0.000, B 0.000, C 0.000 }
gfCNCPoint5[10848] = {X 227.8805, Y 12.1868, Z -7.1667, A 0.000, B 0.000, C 0.000 }
gfCNCPoint5[10849] = {X 227.8802, Y 13.0233, Z -7.1667, A 0.000, B 0.000, C 0.000 }
gfCNCPoint5[10850] = {X 227.7720, Y 13.9490, Z -7.1667, A 0.000, B 0.000, C 0.000 }
gfCNCPoint5[10851] = {X 227.4713, Y 14.8311, Z -7.1667, A 0.000, B 0.000, C 0.000 }
gfCNCPoint5[10852] = {X 226.9915, Y 15.6300, Z -7.1667, A 0.000, B 0.000, C 0.000 }
gfCNCPoint5[10853] = {X 226.3541, Y 16.3100, Z -7.1667, A 0.000, B 0.000, C 0.000 }
gfCNCPoint5[10854] = {X 226.3551, Y 40.8776, Z -7.1667, A 0.000, B 0.000, C 0.000 }
gfCNCPoint5[10855] = {X 226.9988, Y 41.5666, Z -7.1667, A 0.000, B 0.000, C 0.000 }
gfCNCPoint5[10856] = {X 227.4810, Y 42.3769, Z -7.1667, A 0.000, B 0.000, C 0.000 }
gfCNCPoint5[10857] = {X 227.7795, Y 43.2714, Z -7.1667, A 0.000, B 0.000, C 0.000 }
gfCNCPoint5[10858] = {X 227.8805, Y 44.2089, Z -7.1667, A 0.000, B 0.000, C 0.000 }
gfCNCPoint5[10859] = {X 227.8805, Y 45.0000, Z -7.1667, A 0.000, B 0.000, C 0.000 }
gfCNCPoint5[10860] = {X 227.8037, Y 45.8182, Z -7.1667, A 0.000, B 0.000, C 0.000 }
gfCNCPoint5[10861] = {X 227.5762, Y 46.6079, Z -7.1667, A 0.000, B 0.000, C 0.000 }
gfCNCPoint5[10862] = {X 227.2057, Y 47.3415, Z -7.1667, A 0.000, B 0.000, C 0.000 }
gfCNCPoint5[10863] = {X 226.7053, Y 47.9934, Z -7.1667, A 0.000, B 0.000, C 0.000 }
gfCNCPoint5[10864] = {X 227.0571, Y 48.3200, Z -7.1667, A 0.000, B 0.000, C 0.000 }
